// oaksLibrary/fbPushButton
//Funktionsblock för återfjädrande tryckknappar. För tex. förlängd drift aggregat. Om knapp återaktiveras innan tid löpt ut avvaktiveras utgång.
FUNCTION_BLOCK fbPushButton
VAR_INPUT
	bForceIndication : BOOL :=FALSE; //Tvångsstyrning indikering i tryckknapp
	bActiveTrig : BOOL := FALSE; // Läge på aktivering (V-tagg) ändras vid puls in på denna ingång. Är (V-tagg) till går den från och vise versa.
END_VAR

VAR_OUTPUT
	{attribute 'OPC.UA.DA' := '1'}
	V AT %M* : BOOL; //Aktiverad~wp:[trendoptions]i:14400, t:1
	{attribute 'OPC.UA.DA' := '1'}
	CMD AT %Q*: BOOL; //Indikering~wp:[trendoptions]i:14400, t:1
	{attribute 'OPC.UA.DA' := '1'}
	PV1 AT %M* : INT; //Återstående tid~wp:[unit]min[format]0
END_VAR

VAR
	bInput AT %I*: BOOL :=FALSE; //Ingång
	bMode: INT :=0; // Lägesindikering knapp 0=Avaktiverad funktion 1=Aktiverad knapp 2=Återaktiverad knapp (reset)
	bPulse: BOOL :=FALSE; // Startpuls
	tTime: TIME;
	rElapsed: REAL;
	rSetTime: REAL;
	fbResetTon : TON;
	fbTriggerPulse: TP;
	fbActivated: TP;
	fbCounter: CTU;
	fbResetFallingEdge: F_TRIG;	
END_VAR

VAR_INPUT PERSISTENT
	{attribute 'OPC.UA.DA' := '1'}
	SP1 AT %M*: INT :=120; //Frånslagsfördröjning~wp:[unit]min[format]0
	{attribute 'OPC.UA.DA' := '1'}
	M AT %M*: BOOL; //Handkörning~wp:[trendoptions]i:14400, t:1
END_VAR

	IF M THEN
		fbResetTon.IN := TRUE;
		IF fbResetTon.Q THEN
			M := FALSE;
		END_IF
	ELSE
		fbResetTon.IN := FALSE;
	END_IF
	fbResetTon.PT := T#0.5S;
	fbResetTon();

//Startpuls
fbTriggerPulse(IN:= bInput OR M OR bActiveTrig , PT:= T#0.5S , Q=> bPulse, ET=> );

//Återstånde tid
rElapsed := TIME_TO_REAL(fbActivated.ET);
rSetTime := TIME_TO_REAL(fbActivated.PT);
PV1 := REAL_TO_INT((rSetTime - rElapsed)/60000);

//Tidskonvertering till min->ms
tTime := INT_TO_TIME(SP1)*60000;

//Läge på knapp 
fbCounter(
	CU:= bPulse, 
	RESET:= fbCounter.Q OR fbResetFallingEdge.Q, 
	PV:= 2, 
	Q=> , 
	CV=>);

bMode := WORD_TO_INT(fbCounter.CV);

CASE bMode OF
0:
fbActivated.PT := T#0S;
1:
fbActivated.PT := tTime ;	
END_CASE
//Utgång
fbActivated(IN:= bMode=1, PT:=, Q=> V, ET=> );
CMD := V OR bForceIndication;
//Reset av funktion då tid löpt ut
fbResetFallingEdge(CLK:= fbActivated.Q , Q=> );

END_FUNCTION_BLOCK

// oaksLibrary/Regulatorer/Utökade regulatorer/fbAdvSequenceController2Stages
// Pi-regulator 2-sekvens
// För utökad kontroll av reglering:
// bPause fryser regulatorns läge
// bSync synkar regulatorns aktuella sekvens till sitt inställda rSync-värde
// udiInitSwDl är fördröjning innan byte av sekvens vid uppstart (om 0 funkar ej vald startsekvens om PV < SP)
// rSyncSeq[n] är synkvärde för resp sekvens
// rOffValSeq[n] är fast utsignal då bEnable = FALSE
{attribute 'initialize_on_call'}
FUNCTION_BLOCK fbAdvSequenceController2Stages
VAR_INPUT
	bEnable : BOOL; // Aktiverar reglering
	bPause : BOOL := FALSE; // Pausa regulator
	bSync : BOOL := FALSE; // Synkronisera aktuell sekvens till rSync
	udiInitSwDl : UDINT := 5; // Fördröjning för växling av sekvens vid uppstart (minst 1 om startsekvens ska gälla)	
	rProcessValue : REAL; // Aktuellt Ärvärde 
	rSetpoint : REAL; // Aktuellt börvärde. Önskas separat kylbörvärde för kylsekvenser se inputen rCoolSetpoint.
	{attribute 'initialize_on_call'}
	rCoolSetpoint : REFERENCE TO REAL := 0; //Om man önskar ha ett högre börvärde för kylsekvenser lägg denna här så väljs detta på de sekvenser där bActnSequenceX = TRUE. Lämnar man inputen tom körs rSetpoint på både kyl och värmesekvenser.
	iStartSequence : UDINT := 2; //Sekvens där regulator startar
	
	rMinSeq1 : REAL := 0; 
	rMaxSeq1 : REAL := 100; 
	rSyncSeq1 : REAL := 0;	//Synkvärde
	rOffValSeq1 : REAL := 0; //Utgång om ej bEnable
	bActnSequence1 : BOOL; // Gångriktning reglersekvens  (kylsekvens = TRUE)
	bBlockSequence1 : BOOL; // blockera denna sekvens kan användas exempelvis vid nattkyla
	rKpSequence1 : REAL; // Kp
	rKiSequence1 : UDINT; // Ki
	rDiSequence1 : UDINT; // D-tid (Derivata)
	rFDiSequence1 : UDINT; // Filter tid D (Derivata)
	rDzSequence1 : REAL :=0.1; //Dödzon
	
	rMinSeq2 : REAL := 0; 
	rMaxSeq2 : REAL := 100; 
	rSyncSeq2 : REAL := 0;	//Synkvärde
	rOffValSeq2 : REAL := 0; //Utgång om ej bEnable
	bActnSequence2 : BOOL; // Gångriktning reglersekvens  (kylsekvens = TRUE)
	bBlockSequence2 : BOOL; // blockera denna sekvens kan användas exempelvis vid nattkyla
	rKpSequence2 : REAL; // Kp
	rKiSequence2 : UDINT; // Ki
	rDiSequence2 : UDINT; // D-tid (Derivata)
	rFDiSequence2 : UDINT; // Filter tid D (Derivata)
	rDzSequence2 : REAL :=0.1; //Dödzon

	{attribute 'initialize_on_call'}
	rDevLimit : REFERENCE TO REAL := 0;
	{attribute 'pingroup' := 'DeviationAlarm'}
	bBlockHighAlarm : BOOL; // Blockera högtemplarm
	{attribute 'pingroup' := 'DeviationAlarm'}
	bBlockLowAlarm : BOOL; // Blockera lågtemplarm
	{attribute 'pingroup' := 'DeviationAlarm'}
	tAlarmDelay : TIME := T#5S; // larmfördröjning
END_VAR
VAR_OUTPUT
	rOutputSequence1 : REAL;  // regulatorsignal
	rOutputSequence2 : REAL;  // regulatorsignal
	{attribute 'pingroup' := 'DeviationAlarm'}
	bAlarmOutput : BOOL; //larmutgång
END_VAR
VAR
	rDevLimitInternal : REAL;
	fbDevAlarmPV: fbDevAlarm;
	rSetPointSequence1,rSetPointSequence2 : REAL; 	

	rTempMin,rTempMax : REAL; // tempvariabel för blockering av sekvenser 
	fbSeqLink01: Tc3_BA_Common.FB_BA_SeqLink;
	stSeqLink01 : Tc3_BA_Common.ST_BA_SeqLink;
	fbPidSeq: ARRAY[1..2] OF Tc3_BA_Common.FB_BA_SeqCtrl;
	iStartSequenceInternal : UDINT := 2;
	
	fbEdgeEnable : fbEdge;
END_VAR

fbEdgeEnable(anyInput := bEnable);
IF fbEdgeEnable.bEdgeF THEN bSync := TRUE; END_IF	

fbDevAlarmPV(
	tAlarmDelay:=tAlarmDelay , 
	bAutoReset:=TRUE , 
	bAlarmOutput=>bAlarmOutput , 
	bEnable:=bEnable AND mDevAlarmCheck(), 
	rProcessValue:=rProcessValue , 
	rSetPoint:=rSetpoint , 
	rDevLimit:=rDevLimitInternal , 
	bBlockHighAlarm:=bBlockHighAlarm , 
	bBlockLowAlarm:=bBlockLowAlarm );

	IF iStartSequence > 0 AND iStartSequence < 3 THEN
	 iStartSequenceInternal	 := 3 - iStartSequence;
	END_IF;

IF NOT bPause THEN
	fbSeqLink01(
	bEn:= bEnable, 
	udiSttCtrl:=iStartSequenceInternal , 
	udiIniSwiOvrDly_sec:= udiInitSwDl, 
	rX:= rProcessValue, 
	stSeqLink:=stSeqLink01 , 
	udiCurCtrl=> , 
	bSeqActv=> , 
	bNotRead=> , 
	bNoneOp=> , 
	udiRemTiIniSwiOvrDly_sec=> , 
	bErr=> , 
	sErrDescr=> );
	
	IF bBlockSequence1 THEN
		rTempMin := 0;
		rTempMax := 0;
	ELSE
		rTempMin := rMinSeq1;
		rTempMax := rMaxSeq1;
	END_IF
	rSetPointSequence1 := mCoolSetpointCheck(bActnSequence1);
	fbPidSeq[1](
	bEn:=bEnable , 
	rW:= rSetPointSequence1, 
	rX:=rProcessValue , 
	udiOpMode:= , 
	bActn:=bActnSequence1 , 
	rKp:= rKpSequence1, 
	udiTn_ms:=rKiSequence1*1000 , 
	udiTv_ms:=rDiSequence1*1000 , 
	udiTd_ms:=rFDiSequence1*1000 , 
	rYMax:=rTempMax , 
	rYMin:=rTempMin , 
	rNZ:= rDzSequence1, 
	udiCycCl:= , 
	bSync:= bSync, 
	rSync:= rSyncSeq1, 
	rYSeqInit:= rSyncSeq1, 
	udiMyNum:= 2, 
	stSeqLink:=stSeqLink01 , 
	rY=> rOutputSequence1, 
	rE=> , 
	bErr=> , 
	sErrDescr=> );
	
	IF bBlockSequence2 THEN
		rTempMin := 0;
		rTempMax := 0;
	ELSE
		rTempMin := rMinSeq2;
		rTempMax := rMaxSeq2;
	END_IF
	rSetPointSequence2 := mCoolSetpointCheck(bActnSequence2);
	fbPidSeq[2](
	bEn:=bEnable , 
	rW:= rSetPointSequence2, 
	rX:= rProcessValue, 
	udiOpMode:= , 
	bActn:= bActnSequence2, 
	rKp:= rKpSequence2, 
	udiTn_ms:=rKiSequence2*1000 , 
	udiTv_ms:=rDiSequence2*1000  , 
	udiTd_ms:=rFDiSequence2*1000 , 
	rYMax:=rTempMax , 
	rYMin:=rTempMin , 
	rNZ:= rDzSequence2, 
	udiCycCl:= , 
	bSync:= bSync, 
	rSync:= rSyncSeq2, 
	rYSeqInit:= rSyncSeq2, 
	udiMyNum:= 1, 
	stSeqLink:= stSeqLink01, 
	rY=> rOutputSequence2, 
	rE=> , 
	bErr=> , 
	sErrDescr=> );
	
	bSync := FALSE;	
END_IF;

IF NOT bEnable THEN
	rOutputSequence1 := rOffValSeq1;
	rOutputSequence2 := rOffValSeq2;
END_IF

// Publik metod för att kolla ifall det finns någon kylsekvens i regleringen. Kan exempelvis användas för att blockera högavvikelselarm vid hög utetemperatur då kylsekvens saknas.
METHOD PUBLIC mContainsCoolingSequence : BOOL
mContainsCoolingSequence := bActnSequence1 OR bActnSequence2;
END_METHOD

// Metod för att kolla ifall det är en kylsekvens och om det i sådant fall är något knutet på rCoolSetpoint
METHOD PRIVATE mCoolSetpointCheck : REAL // Valt börvärde
VAR_INPUT
	bActn : BOOL; // Koll av gångriktning
END_VAR
IF NOT bActn THEN
	mCoolSetpointCheck := rSetpoint;
ELSE
	IF __ISVALIDREF(rCoolSetpoint) THEN 
		mCoolSetpointCheck := rCoolSetpoint;
	ELSE
		mCoolSetpointCheck := rSetpoint;
	END_IF
END_IF
END_METHOD

// Kolla ifall något är knutet på inputen rDevLimit. Är inget knutet där inaktiveras avvikelselarmet.
METHOD PRIVATE mDevAlarmCheck : BOOL // Valt börvärde
IF __ISVALIDREF(rDevLimit) THEN 
	mDevAlarmCheck := TRUE;
	rDevLimitInternal := rDevLimit;
ELSE
	mDevAlarmCheck := FALSE;
END_IF
END_METHOD

END_FUNCTION_BLOCK

// oaksLibrary/Regulatorer/Utökade regulatorer/fbAdvSequenceController3Stages
// Pi-regulator 3-sekvens
// För utökad kontroll av reglering:
// bPause fryser regulatorns läge
// bSync synkar regulatorns aktuella sekvens till sitt inställda rSync-värde
// udiInitSwDl är fördröjning innan byte av sekvens vid uppstart (om 0 funkar ej vald startsekvens om PV < SP)
// rSyncSeq[n] är synkvärde för resp sekvens
// rOffValSeq[n] är fast utsignal då bEnable = FALSE
{attribute 'initialize_on_call'}
FUNCTION_BLOCK fbAdvSequenceController3Stages
VAR_INPUT
	bEnable : BOOL; // Aktiverar reglering (toggla för att reset:a regulator)
	bPause : BOOL := FALSE; // Pausa regulator
	bSync : BOOL := FALSE; // Synkronisera aktuell sekvens till rSync
	udiInitSwDl : UDINT := 5; // Fördröjning för växling av sekvens vid uppstart (minst 1 om startsekvens ska gälla)	
	rProcessValue : REAL; // Aktuellt Ärvärde 
	rSetpoint : REAL; // Aktuellt börvärde. Önskas separat kylbörvärde för kylsekvenser se inputen rCoolSetpoint.
	{attribute 'initialize_on_call'}
	rCoolSetpoint : REFERENCE TO REAL; //Om man önskar ha ett högre börvärde för kylsekvenser lägg denna här så väljs detta på de sekvenser där bActnSequenceX = TRUE. Lämnar man inputen tom körs rSetpoint på både kyl och värmesekvenser.
	iStartSequence : UDINT :=3; //Sekvens där regulator startar
	
	rMinSeq1 : REAL := 0;	//Min utsignal
	rMaxSeq1 : REAL := 100;	//Max utsignal
	rSyncSeq1 : REAL := 0;	//Synkvärde
	rOffValSeq1 : REAL := 0; //Utgång om ej bEnable
	bActnSequence1 : BOOL; // Gångriktning reglersekvens  (kylsekvens = TRUE)
	bBlockSequence1 : BOOL; // blockera denna sekvens kan användas exempelvis vid nattkyla
	rKpSequence1 : REAL; // Kp
	rKiSequence1 : UDINT; // Ki
	rDiSequence1 : UDINT; // D-tid (Derivata)
	rFDiSequence1 : UDINT; // Filter tid D (Derivata)
	rDzSequence1 : REAL :=0.1; //Dödzon
	
	rMinSeq2 : REAL := 0; 
	rMaxSeq2 : REAL := 100;
	rSyncSeq2 : REAL := 0;
	rOffValSeq2 : REAL := 0; //Utgång om ej bEnable
	bActnSequence2 : BOOL; // Gångriktning reglersekvens  (kylsekvens = TRUE)
	bBlockSequence2 : BOOL; // blockera denna sekvens kan användas exempelvis vid nattkyla
	rKpSequence2 : REAL; // Kp
	rKiSequence2 : UDINT; // Ki
	rDiSequence2 : UDINT; // D-tid (Derivata)
	rFDiSequence2 : UDINT; // Filter tid D (Derivata)
	rDzSequence2 : REAL :=0.1; //Dödzon
	
	rMinSeq3 : REAL := 0; 
	rMaxSeq3 : REAL := 100;
	rSyncSeq3 : REAL := 0;
	rOffValSeq3 : REAL := 0; //Utgång om ej bEnable
	bActnSequence3 : BOOL; // Gångriktning reglersekvens  (kylsekvens = TRUE)
	bBlockSequence3 : BOOL; // blockera denna sekvens kan användas exempelvis vid nattkyla
	rKpSequence3 : REAL; // Kp
	rKiSequence3 : UDINT; // Ki
	rDiSequence3 : UDINT; // D-tid (Derivata)
	rFDiSequence3 : UDINT; // Filter tid D (Derivata)
	rDzSequence3 : REAL :=0.1; //Dödzon
	
	{attribute 'pingroup' := 'DeviationAlarm'}
	{attribute 'initialize_on_call'}
	rDevLimit : REFERENCE TO REAL := 0;
	{attribute 'pingroup' := 'DeviationAlarm'}
	bBlockHighAlarm : BOOL; // Blockera högtemplarm
	{attribute 'pingroup' := 'DeviationAlarm'}
	bBlockLowAlarm : BOOL; // Blockera lågtemplarm
	{attribute 'pingroup' := 'DeviationAlarm'}
	tAlarmDelay : TIME := T#5S; // larmfördröjning
END_VAR
VAR_OUTPUT
	rOutputSequence1 : REAL;  // regulatorsignal
	rOutputSequence2 : REAL;  // regulatorsignal
	rOutputSequence3 : REAL;  // regulatorsignal
	{attribute 'pingroup' := 'DeviationAlarm'}
	bAlarmOutput : BOOL; //larmutgång
END_VAR
VAR
	rDevLimitInternal : REAL;
	fbDevAlarmPV: fbDevAlarm;
	rSetPointSequence1,rSetPointSequence2,rSetPointSequence3 : REAL; 		

	rTempMin,rTempMax : REAL; // tempvariabel för blockering av sekvenser 
	fbSeqLink01: Tc3_BA_Common.FB_BA_SeqLink;
	stSeqLink01 : Tc3_BA_Common.ST_BA_SeqLink;
	fbPidSeq: ARRAY[1..3] OF Tc3_BA_Common.FB_BA_SeqCtrl;
	iStartSequenceInternal : UDINT := 3;
	
	fbEdgeEnable : fbEdge;
END_VAR

fbEdgeEnable(anyInput := bEnable);
IF fbEdgeEnable.bEdgeF THEN bSync := TRUE; END_IF

fbDevAlarmPV(
tAlarmDelay:=tAlarmDelay , 
bAutoReset:=TRUE , 
bAlarmOutput=>bAlarmOutput , 
bEnable:=bEnable AND mDevAlarmCheck(), 
rProcessValue:=rProcessValue , 
rSetPoint:=rSetpoint , 
rDevLimit:=rDevLimitInternal , 
bBlockHighAlarm:=bBlockHighAlarm , 
bBlockLowAlarm:=bBlockLowAlarm );

IF iStartSequence > 0 AND iStartSequence < 4 THEN
 iStartSequenceInternal	 := 4 - iStartSequence;
END_IF;
		
IF NOT bPause THEN	
	fbSeqLink01(
	bEn:= bEnable, 
	udiSttCtrl:= iStartSequenceInternal, 
	udiIniSwiOvrDly_sec:= udiInitSwDl, 
	rX:= rProcessValue, 
	stSeqLink:=stSeqLink01 , 
	udiCurCtrl=> , 
	bSeqActv=> , 
	bNotRead=> , 
	bNoneOp=> , 
	udiRemTiIniSwiOvrDly_sec=> , 
	bErr=> , 
	sErrDescr=> );
	
	IF bBlockSequence1 THEN
		rTempMin := 0;
		rTempMax := 0;
	ELSE
		rTempMin := rMinSeq1;
		rTempMax := rMaxSeq1;
	END_IF
	rSetPointSequence1 := mCoolSetpointCheck(bActnSequence1);
	fbPidSeq[1](
	bEn:=bEnable , 
	rW:= rSetPointSequence1, 
	rX:=rProcessValue , 
	udiOpMode:= , 
	bActn:=bActnSequence1 , 
	rKp:= rKpSequence1, 
	udiTn_ms:=rKiSequence1*1000 , 
	udiTv_ms:=rDiSequence1*1000 , 
	udiTd_ms:=rFDiSequence1*1000 , 
	rYMax:=rTempMax , 
	rYMin:= rTempMin, 
	rNZ:= rDzSequence1, 
	udiCycCl:= , 
	bSync:= bSync, 
	rSync:= rSyncSeq1, 
	rYSeqInit:= rSyncSeq1, 
	udiMyNum:= 3, 
	stSeqLink:=stSeqLink01 , 
	rY=> rOutputSequence1, 
	rE=> , 
	bErr=> , 
	sErrDescr=> );
	
	IF bBlockSequence2 THEN
		rTempMin := 0;
		rTempMax := 0;
	ELSE
		rTempMin := rMinSeq2;
		rTempMax := rMaxSeq2;
	END_IF
	rSetPointSequence2 := mCoolSetpointCheck(bActnSequence2);
	fbPidSeq[2](
	bEn:=bEnable , 
	rW:= rSetPointSequence2, 
	rX:= rProcessValue, 
	udiOpMode:= , 
	bActn:= bActnSequence2, 
	rKp:= rKpSequence2, 
	udiTn_ms:=rKiSequence2*1000 , 
	udiTv_ms:=rDiSequence2*1000 , 
	udiTd_ms:=rFDiSequence2*1000 , 
	rYMax:= rTempMax, 
	rYMin:=rTempMin , 
	rNZ:= rDzSequence2, 
	udiCycCl:= , 
	bSync:= bSync,  
	rSync:= rSyncSeq2, 
	rYSeqInit:= rSyncSeq2, 
	udiMyNum:= 2, 
	stSeqLink:= stSeqLink01, 
	rY=> rOutputSequence2, 
	rE=> , 
	bErr=> , 
	sErrDescr=> );
	
	IF bBlockSequence3 THEN
		rTempMin := 0;
		rTempMax := 0;
	ELSE
		rTempMin := rMinSeq3;
		rTempMax := rMaxSeq3;
	END_IF
	rSetPointSequence3 := mCoolSetpointCheck(bActnSequence3);
	fbPidSeq[3](
	bEn:=bEnable , 
	rW:= rSetPointSequence3, 
	rX:= rProcessValue, 
	udiOpMode:= , 
	bActn:= bActnSequence3, 
	rKp:= rKpSequence3, 
	udiTn_ms:=rKiSequence3*1000 , 
	udiTv_ms:=rDiSequence3*1000 , 
	udiTd_ms:=rFDiSequence3*1000 , 
	rYMax:=rTempMax , 
	rYMin:= rTempMin, 
	rNZ:= rDzSequence3, 
	udiCycCl:= , 
	bSync:= bSync, 
	rSync:= rSyncSeq3, 
	rYSeqInit:= rSyncSeq3, 
	udiMyNum:= 1, 
	stSeqLink:= stSeqLink01, 
	rY=> rOutputSequence3, 
	rE=> , 
	bErr=> , 
	sErrDescr=> );
	
	bSync := FALSE;	
END_IF;

IF NOT bEnable THEN
	rOutputSequence1 := rOffValSeq1;
	rOutputSequence2 := rOffValSeq2;
	rOutputSequence3 := rOffValSeq3;
END_IF

// Publik metod för att kolla ifall det finns någon kylsekvens i regleringen. Kan exempelvis användas för att blockera högavvikelselarm vid hög utetemperatur då kylsekvens saknas.
METHOD PUBLIC mContainsCoolingSequence : BOOL
mContainsCoolingSequence := bActnSequence1 OR bActnSequence2 OR bActnSequence3;
END_METHOD

// Metod för att kolla ifall det är en kylsekvens och om det i sådant fall är något knutet på rCoolSetpoint
METHOD PRIVATE mCoolSetpointCheck : REAL // Valt börvärde
VAR_INPUT
	bActn : BOOL; // Koll av gångriktning
END_VAR
IF NOT bActn THEN
	mCoolSetpointCheck := rSetpoint;
ELSE
	IF __ISVALIDREF(rCoolSetpoint) THEN 
		mCoolSetpointCheck := rCoolSetpoint;
	ELSE
		mCoolSetpointCheck := rSetpoint;
	END_IF
END_IF
END_METHOD

// Kolla ifall något är knutet på inputen rDevLimit. Är inget knutet där inaktiveras avvikelselarmet.
METHOD PRIVATE mDevAlarmCheck : BOOL // Valt börvärde
IF __ISVALIDREF(rDevLimit) THEN 
	mDevAlarmCheck := TRUE;
	rDevLimitInternal := rDevLimit;
ELSE
	mDevAlarmCheck := FALSE;
END_IF
END_METHOD

END_FUNCTION_BLOCK

// oaksLibrary/Regulatorer/Utökade regulatorer/fbAdvSequenceController4Stages
// Pi-regulator 4-sekvens
// För utökad kontroll av reglering:
// bPause fryser regulatorns läge
// bSync synkar regulatorns aktuella sekvens till sitt inställda rSync-värde
// udiInitSwDl är fördröjning innan byte av sekvens vid uppstart (om 0 funkar ej vald startsekvens om PV < SP)
// rSyncSeq[n] är synkvärde för resp sekvens
// rOffValSeq[n] är fast utsignal då bEnable = FALSE
{attribute 'initialize_on_call'}
FUNCTION_BLOCK fbAdvSequenceController4Stages
VAR_INPUT
	bEnable : BOOL; // Aktiverar reglering (toggla för att reset:a regulator)
	bPause : BOOL := FALSE; // Pausa regulator
	bSync : BOOL := FALSE; // Synkronisera aktuell sekvens till rSync
	udiInitSwDl : UDINT := 5; // Fördröjning för växling av sekvens vid uppstart (minst 1 om startsekvens ska gälla)	
	rProcessValue : REAL; // Aktuellt Ärvärde 
	rSetpoint : REAL; // Aktuellt börvärde. Önskas separat kylbörvärde för kylsekvenser se inputen rCoolSetpoint.
	{attribute 'initialize_on_call'}
	rCoolSetpoint : REFERENCE TO REAL; //Om man önskar ha ett högre börvärde för kylsekvenser lägg denna här så väljs detta på de sekvenser där bActnSequenceX = TRUE. Lämnar man inputen tom körs rSetpoint på både kyl och värmesekvenser.
	iStartSequence : UDINT :=3; //Sekvens där regulator startar
	
	rMinSeq1 : REAL := 0;	//Min utsignal
	rMaxSeq1 : REAL := 100;	//Max utsignal
	rSyncSeq1 : REAL := 0;	//Synkvärde
	rOffValSeq1 : REAL := 0; //Utgång om ej bEnable
	bActnSequence1 : BOOL; // Gångriktning reglersekvens  (kylsekvens = TRUE)
	bBlockSequence1 : BOOL; // blockera denna sekvens kan användas exempelvis vid nattkyla
	rKpSequence1 : REAL; // Kp
	rKiSequence1 : UDINT; // Ki
	rDiSequence1 : UDINT; // D-tid (Derivata)
	rFDiSequence1 : UDINT; // Filter tid D (Derivata)
	rDzSequence1 : REAL :=0.1; //Dödzon
	
	rMinSeq2 : REAL := 0; 
	rMaxSeq2 : REAL := 100;
	rSyncSeq2 : REAL := 0;
	rOffValSeq2 : REAL := 0; //Utgång om ej bEnable
	bActnSequence2 : BOOL; // Gångriktning reglersekvens  (kylsekvens = TRUE)
	bBlockSequence2 : BOOL; // blockera denna sekvens kan användas exempelvis vid nattkyla
	rKpSequence2 : REAL; // Kp
	rKiSequence2 : UDINT; // Ki
	rDiSequence2 : UDINT; // D-tid (Derivata)
	rFDiSequence2 : UDINT; // Filter tid D (Derivata)
	rDzSequence2 : REAL :=0.1; //Dödzon
	
	rMinSeq3 : REAL := 0; 
	rMaxSeq3 : REAL := 100;
	rSyncSeq3 : REAL := 0;
	rOffValSeq3 : REAL := 0; //Utgång om ej bEnable
	bActnSequence3 : BOOL; // Gångriktning reglersekvens  (kylsekvens = TRUE)
	bBlockSequence3 : BOOL; // blockera denna sekvens kan användas exempelvis vid nattkyla
	rKpSequence3 : REAL; // Kp
	rKiSequence3 : UDINT; // Ki
	rDiSequence3 : UDINT; // D-tid (Derivata)
	rFDiSequence3 : UDINT; // Filter tid D (Derivata)
	rDzSequence3 : REAL :=0.1; //Dödzon
	
	rMinSeq4 : REAL := 0; 
	rMaxSeq4 : REAL := 100;
	rSyncSeq4 : REAL := 0;
	rOffValSeq4 : REAL := 0; //Utgång om ej bEnable
	bActnSequence4 : BOOL; // Gångriktning reglersekvens  (kylsekvens = TRUE)
	bBlockSequence4 : BOOL; // blockera denna sekvens kan användas exempelvis vid nattkyla
	rKpSequence4 : REAL; // Kp
	rKiSequence4 : UDINT; // Ki
	rDiSequence4 : UDINT; // D-tid (Derivata)
	rFDiSequence4 : UDINT; // Filter tid D (Derivata)
	rDzSequence4 : REAL :=0.1; //Dödzon
	
	{attribute 'pingroup' := 'DeviationAlarm'}
	{attribute 'initialize_on_call'}
	rDevLimit : REFERENCE TO REAL := 0;
	{attribute 'pingroup' := 'DeviationAlarm'}
	bBlockHighAlarm : BOOL; // Blockera högtemplarm
	{attribute 'pingroup' := 'DeviationAlarm'}
	bBlockLowAlarm : BOOL; // Blockera lågtemplarm
	{attribute 'pingroup' := 'DeviationAlarm'}
	tAlarmDelay : TIME := T#5S; // larmfördröjning
END_VAR
VAR_OUTPUT
	rY : REAL; // Utsignal huvudregulator
	rOutputSequence1 : REAL;  // regulatorsignal
	rOutputSequence2 : REAL;  // regulatorsignal
	rOutputSequence3 : REAL;  // regulatorsignal
	rOutputSequence4 : REAL;  // regulatorsignal
	{attribute 'pingroup' := 'DeviationAlarm'}
	bAlarmOutput : BOOL; //larmutgång
END_VAR
VAR
	rDevLimitInternal : REAL;
	fbDevAlarmPV: fbDevAlarm;
	rSetPointSequence1,rSetPointSequence2,rSetPointSequence3,rSetPointSequence4 : REAL; 	
	rTempMin,rTempMax : REAL; // tempvariabel för blockering av sekvenser 
	fbSeqLink01: Tc3_BA_Common.FB_BA_SeqLink;
	stSeqLink01 : Tc3_BA_Common.ST_BA_SeqLink;
	fbPidSeq: ARRAY[1..4] OF Tc3_BA_Common.FB_BA_SeqCtrl;
	iStartSequenceInternal : UDINT := 3;
	
	fbEdgeEnable : fbEdge;
END_VAR

fbEdgeEnable(anyInput := bEnable);
IF fbEdgeEnable.bEdgeF THEN bSync := TRUE; END_IF

	fbDevAlarmPV(
	tAlarmDelay:=tAlarmDelay , 
	bAutoReset:=TRUE , 
	bAlarmOutput=>bAlarmOutput , 
	bEnable:=bEnable AND mDevAlarmCheck(), 
	rProcessValue:=rProcessValue , 
	rSetPoint:=rSetpoint , 
	rDevLimit:=rDevLimitInternal , 
	bBlockHighAlarm:=bBlockHighAlarm , 
	bBlockLowAlarm:=bBlockLowAlarm );

	IF iStartSequence > 0 AND iStartSequence < 5 THEN
	 iStartSequenceInternal	 := 5 - iStartSequence;
	END_IF;
		
IF NOT bPause THEN		
	fbSeqLink01(
	bEn:= bEnable, 
	udiSttCtrl:= iStartSequenceInternal, 
	udiIniSwiOvrDly_sec:= udiInitSwDl, 
	rX:= rProcessValue, 
	stSeqLink:=stSeqLink01 , 
	udiCurCtrl=> , 
	bSeqActv=> , 
	bNotRead=> , 
	bNoneOp=> , 
	udiRemTiIniSwiOvrDly_sec=> , 
	bErr=> , 
	sErrDescr=> );
		
	IF bBlockSequence1 THEN
		rTempMin := 0;
		rTempMax := 0;
	ELSE
		rTempMin := rMinSeq1;
		rTempMax := rMaxSeq1;
	END_IF
	rSetPointSequence1 := mCoolSetpointCheck(bActnSequence1);
	fbPidSeq[1](
	bEn:=bEnable , 
	rW:= rSetPointSequence1, 
	rX:=rProcessValue , 
	udiOpMode:= , 
	bActn:=bActnSequence1 , 
	rKp:= rKpSequence1, 
	udiTn_ms:=rKiSequence1*1000 , 
	udiTv_ms:=rDiSequence1*1000 , 
	udiTd_ms:=rFDiSequence1*1000 , 
	rYMax:=rTempMax , 
	rYMin:=rTempMin, 
	rNZ:= rDzSequence1, 
	udiCycCl:= , 
	bSync:= bSync, 
	rSync:= rSyncSeq1, 
	rYSeqInit:= rSyncSeq1, 
	udiMyNum:= 4, 
	stSeqLink:=stSeqLink01 , 
	rY=> rOutputSequence1, 
	rE=> , 
	bErr=> , 
	sErrDescr=> );
	
	IF bBlockSequence2 THEN
		rTempMin := 0;
		rTempMax := 0;
	ELSE
		rTempMin := rMinSeq2;
		rTempMax := rMaxSeq2;
	END_IF
	rSetPointSequence2 := mCoolSetpointCheck(bActnSequence2);
	fbPidSeq[2](
	bEn:=bEnable , 
	rW:= rSetPointSequence2, 
	rX:= rProcessValue, 
	udiOpMode:= , 
	bActn:= bActnSequence2, 
	rKp:= rKpSequence2, 
	udiTn_ms:=rKiSequence2*1000 , 
	udiTv_ms:=rDiSequence2*1000 , 
	udiTd_ms:=rFDiSequence2*1000 , 
	rYMax:= rTempMax, 
	rYMin:=rTempMin , 
	rNZ:= rDzSequence2, 
	udiCycCl:= , 
	bSync:= bSync, 
	rSync:= rSyncSeq2, 
	rYSeqInit:= rSyncSeq2, 
	udiMyNum:= 3, 
	stSeqLink:= stSeqLink01, 
	rY=> rOutputSequence2, 
	rE=> , 
	bErr=> , 
	sErrDescr=> );
	
	IF bBlockSequence3 THEN
		rTempMin := 0;
		rTempMax := 0;
	ELSE
		rTempMin := rMinSeq3;
		rTempMax := rMaxSeq3;
	END_IF
	rSetPointSequence3 := mCoolSetpointCheck(bActnSequence3);
	fbPidSeq[3](
	bEn:=bEnable , 
	rW:= rSetPointSequence3, 
	rX:= rProcessValue, 
	udiOpMode:= , 
	bActn:= bActnSequence3, 
	rKp:= rKpSequence3, 
	udiTn_ms:=rKiSequence3*1000 , 
	udiTv_ms:=rDiSequence3*1000 , 
	udiTd_ms:=rFDiSequence3*1000 , 
	rYMax:=rTempMax , 
	rYMin:= rTempMin, 
	rNZ:= rDzSequence3, 
	udiCycCl:= , 
	bSync:= bSync, 
	rSync:= rSyncSeq3, 
	rYSeqInit:= rSyncSeq3, 
	udiMyNum:= 2, 
	stSeqLink:= stSeqLink01, 
	rY=> rOutputSequence3, 
	rE=> , 
	bErr=> , 
	sErrDescr=> );
	
	IF bBlockSequence4 THEN
		rTempMin := 0;
		rTempMax := 0;
	ELSE
		rTempMin := rMinSeq4;
		rTempMax := rMaxSeq4;
	END_IF
	rSetPointSequence4 := mCoolSetpointCheck(bActnSequence4);
	fbPidSeq[4](
	bEn:=bEnable , 
	rW:= rSetPointSequence4, 
	rX:= rProcessValue, 
	udiOpMode:= , 
	bActn:= bActnSequence4, 
	rKp:= rKpSequence4, 
	udiTn_ms:=rKiSequence4*1000 , 
	udiTv_ms:=rDiSequence4*1000 , 
	udiTd_ms:=rFDiSequence4*1000 , 
	rYMax:=rTempMax , 
	rYMin:= rTempMin, 
	rNZ:= rDzSequence4, 
	udiCycCl:= , 
	bSync:= bSync, 
	rSync:= rSyncSeq4, 
	rYSeqInit:= rSyncSeq4, 
	udiMyNum:= 1, 
	stSeqLink:= stSeqLink01, 
	rY=> rOutputSequence4, 
	rE=> , 
	bErr=> , 
	sErrDescr=> );
	
	bSync := FALSE;	
END_IF

IF NOT bEnable THEN
	rOutputSequence1 := rOffValSeq1;
	rOutputSequence2 := rOffValSeq2;
	rOutputSequence3 := rOffValSeq3;
	rOutputSequence4 := rOffValSeq4;
END_IF

// Publik metod för att kolla ifall det finns någon kylsekvens i regleringen. Kan exempelvis användas för att blockera högavvikelselarm vid hög utetemperatur då kylsekvens saknas.
METHOD PUBLIC mContainsCoolingSequence : BOOL
mContainsCoolingSequence := bActnSequence1 OR bActnSequence2 OR bActnSequence3 OR bActnSequence4;
END_METHOD

// Metod för att kolla ifall det är en kylsekvens och om det i sådant fall är något knutet på rCoolSetpoint
METHOD PRIVATE mCoolSetpointCheck : REAL // Valt börvärde
VAR_INPUT
	bActn : BOOL; // Koll av gångriktning
END_VAR
IF NOT bActn THEN
	mCoolSetpointCheck := rSetpoint;
ELSE
	IF __ISVALIDREF(rCoolSetpoint) THEN 
		mCoolSetpointCheck := rCoolSetpoint;
	ELSE
		mCoolSetpointCheck := rSetpoint;
	END_IF
END_IF
END_METHOD

// Kolla ifall något är knutet på inputen rDevLimit. Är inget knutet där inaktiveras avvikelselarmet.
METHOD PRIVATE mDevAlarmCheck : BOOL // Valt börvärde
IF __ISVALIDREF(rDevLimit) THEN 
	mDevAlarmCheck := TRUE;
	rDevLimitInternal := rDevLimit;
ELSE
	mDevAlarmCheck := FALSE;
END_IF
END_METHOD

END_FUNCTION_BLOCK

// oaksLibrary/Regulatorer/Utökade regulatorer/fbAdvSequenceController5Stages
// Pi-regulator 5-sekvens
// För utökad kontroll av reglering:
// bPause fryser regulatorns läge
// bSync synkar regulatorns aktuella sekvens till sitt inställda rSync-värde
// udiInitSwDl är fördröjning innan byte av sekvens vid uppstart (om 0 funkar ej vald startsekvens om PV < SP)
// rSyncSeq[n] är synkvärde för resp sekvens
// rOffValSeq[n] är fast utsignal då bEnable = FALSE
{attribute 'initialize_on_call'}
FUNCTION_BLOCK fbAdvSequenceController5Stages
VAR_INPUT
	bEnable : BOOL; // Aktiverar reglering (toggla för att reset:a regulator)
	bPause : BOOL := FALSE; // Pausa regulator
	bSync : BOOL := FALSE; // Synkronisera aktuell sekvens till rSync
	udiInitSwDl : UDINT := 5; // Fördröjning för växling av sekvens vid uppstart (minst 1 om startsekvens ska gälla)	
	rProcessValue : REAL; // Aktuellt Ärvärde 
	rSetpoint : REAL; // Aktuellt börvärde. Önskas separat kylbörvärde för kylsekvenser se inputen rCoolSetpoint.
	{attribute 'initialize_on_call'}
	rCoolSetpoint : REFERENCE TO REAL; //Om man önskar ha ett högre börvärde för kylsekvenser lägg denna här så väljs detta på de sekvenser där bActnSequenceX = TRUE. Lämnar man inputen tom körs rSetpoint på både kyl och värmesekvenser.
	iStartSequence : UDINT :=3; //Sekvens där regulator startar
	
	rMinSeq1 : REAL := 0;	//Min utsignal
	rMaxSeq1 : REAL := 100;	//Max utsignal
	rSyncSeq1 : REAL := 0;	//Synkvärde
	rOffValSeq1 : REAL := 0; //Utgång om ej bEnable
	bActnSequence1 : BOOL; // Gångriktning reglersekvens  (kylsekvens = TRUE)
	bBlockSequence1 : BOOL; // blockera denna sekvens kan användas exempelvis vid nattkyla
	rKpSequence1 : REAL; // Kp
	rKiSequence1 : UDINT; // Ki
	rDiSequence1 : UDINT; // D-tid (Derivata)
	rFDiSequence1 : UDINT; // Filter tid D (Derivata)
	rDzSequence1 : REAL :=0.1; //Dödzon
	
	rMinSeq2 : REAL := 0; 
	rMaxSeq2 : REAL := 100;
	rSyncSeq2 : REAL := 0;
	rOffValSeq2 : REAL := 0; //Utgång om ej bEnable
	bActnSequence2 : BOOL; // Gångriktning reglersekvens  (kylsekvens = TRUE)
	bBlockSequence2 : BOOL; // blockera denna sekvens kan användas exempelvis vid nattkyla
	rKpSequence2 : REAL; // Kp
	rKiSequence2 : UDINT; // Ki
	rDiSequence2 : UDINT; // D-tid (Derivata)
	rFDiSequence2 : UDINT; // Filter tid D (Derivata)
	rDzSequence2 : REAL :=0.1; //Dödzon
	
	rMinSeq3 : REAL := 0; 
	rMaxSeq3 : REAL := 100;
	rSyncSeq3 : REAL := 0;
	rOffValSeq3 : REAL := 0; //Utgång om ej bEnable
	bActnSequence3 : BOOL; // Gångriktning reglersekvens  (kylsekvens = TRUE)
	bBlockSequence3 : BOOL; // blockera denna sekvens kan användas exempelvis vid nattkyla
	rKpSequence3 : REAL; // Kp
	rKiSequence3 : UDINT; // Ki
	rDiSequence3 : UDINT; // D-tid (Derivata)
	rFDiSequence3 : UDINT; // Filter tid D (Derivata)
	rDzSequence3 : REAL :=0.1; //Dödzon
	
	rMinSeq4 : REAL := 0; 
	rMaxSeq4 : REAL := 100;
	rSyncSeq4 : REAL := 0;	//Synkvärde
	rOffValSeq4 : REAL := 0; //Utgång om ej bEnable
	bActnSequence4 : BOOL; // Gångriktning reglersekvens  (kylsekvens = TRUE)
	bBlockSequence4 : BOOL; // blockera denna sekvens kan användas exempelvis vid nattkyla
	rKpSequence4 : REAL; // Kp
	rKiSequence4 : UDINT; // Ki
	rDiSequence4 : UDINT; // D-tid (Derivata)
	rFDiSequence4 : UDINT; // Filter tid D (Derivata)
	rDzSequence4 : REAL :=0.1; //Dödzon
	
	rMinSeq5 : REAL := 0; 
	rMaxSeq5 : REAL := 100;
	rSyncSeq5 : REAL := 0;	//Synkvärde
	rOffValSeq5 : REAL := 0; //Utgång om ej bEnable
	bActnSequence5 : BOOL; // Gångriktning reglersekvens  (kylsekvens = TRUE)
	bBlockSequence5 : BOOL; // blockera denna sekvens kan användas exempelvis vid nattkyla
	rKpSequence5 : REAL; // Kp
	rKiSequence5 : UDINT; // Ki
	rDiSequence5 : UDINT; // D-tid (Derivata)
	rFDiSequence5 : UDINT; // Filter tid D (Derivata)
	rDzSequence5 : REAL :=0.1; //Dödzon
	
	{attribute 'pingroup' := 'DeviationAlarm'}
	{attribute 'initialize_on_call'}
	rDevLimit : REFERENCE TO REAL := 0;
	{attribute 'pingroup' := 'DeviationAlarm'}
	bBlockHighAlarm : BOOL; // Blockera högtemplarm
	{attribute 'pingroup' := 'DeviationAlarm'}
	bBlockLowAlarm : BOOL; // Blockera lågtemplarm
	{attribute 'pingroup' := 'DeviationAlarm'}
	tAlarmDelay : TIME := T#5S; // larmfördröjning
END_VAR
VAR_OUTPUT
	rY : REAL; // Utsignal huvudregulator
	rOutputSequence1 : REAL;  // regulatorsignal
	rOutputSequence2 : REAL;  // regulatorsignal
	rOutputSequence3 : REAL;  // regulatorsignal
	rOutputSequence4 : REAL;  // regulatorsignal
	rOutputSequence5 : REAL;  // regulatorsignal
	{attribute 'pingroup' := 'DeviationAlarm'}
	bAlarmOutput : BOOL; //larmutgång
END_VAR
VAR
	rDevLimitInternal : REAL;
	fbDevAlarmPV: fbDevAlarm;
	rSetPointSequence1,rSetPointSequence2,rSetPointSequence3,rSetPointSequence4,rSetPointSequence5 : REAL; 	
	rTempMin,rTempMax : REAL; // tempvariabel för blockering av sekvenser 
	fbSeqLink01: Tc3_BA_Common.FB_BA_SeqLink;
	stSeqLink01 : Tc3_BA_Common.ST_BA_SeqLink;
	fbPidSeq: ARRAY[1..5] OF Tc3_BA_Common.FB_BA_SeqCtrl;
	iStartSequenceInternal : UDINT := 3;
	
	fbEdgeEnable : fbEdge;
END_VAR

fbEdgeEnable(anyInput := bEnable);
IF fbEdgeEnable.bEdgeF THEN bSync := TRUE; END_IF

fbDevAlarmPV(
	tAlarmDelay:=tAlarmDelay , 
	bAutoReset:=TRUE , 
	bAlarmOutput=>bAlarmOutput , 
	bEnable:=bEnable AND mDevAlarmCheck() , 
	rProcessValue:=rProcessValue , 
	rSetPoint:=rSetpoint , 
	rDevLimit:=rDevLimitInternal , 
	bBlockHighAlarm:=bBlockHighAlarm , 
	bBlockLowAlarm:=bBlockLowAlarm );

	IF iStartSequence > 0 AND iStartSequence < 5 THEN
	 iStartSequenceInternal	 := 5 - iStartSequence;
	END_IF;
		
IF NOT bPause THEN		
	fbSeqLink01(
	bEn:= bEnable, 
	udiSttCtrl:= iStartSequenceInternal, 
	udiIniSwiOvrDly_sec:= udiInitSwDl, 
	rX:= rProcessValue, 
	stSeqLink:=stSeqLink01 , 
	udiCurCtrl=> , 
	bSeqActv=> , 
	bNotRead=> , 
	bNoneOp=> , 
	udiRemTiIniSwiOvrDly_sec=> , 
	bErr=> , 
	sErrDescr=> );
		
	IF bBlockSequence1 THEN
		rTempMin := 0;
		rTempMax := 0;
	ELSE
		rTempMin := rMinSeq1;
		rTempMax := rMaxSeq1;
	END_IF
	rSetPointSequence1 := mCoolSetpointCheck(bActnSequence1);
	fbPidSeq[1](
	bEn:=bEnable , 
	rW:= rSetPointSequence1, 
	rX:=rProcessValue , 
	udiOpMode:= , 
	bActn:=bActnSequence1 , 
	rKp:= rKpSequence1, 
	udiTn_ms:=rKiSequence1*1000 , 
	udiTv_ms:=rDiSequence1*1000 , 
	udiTd_ms:=rFDiSequence1*1000 , 
	rYMax:=rTempMax , 
	rYMin:=rTempMin, 
	rNZ:= rDzSequence1, 
	udiCycCl:= , 
	bSync:= bSync, 
	rSync:= rSyncSeq1, 
	rYSeqInit:= rSyncSeq1, 
	udiMyNum:= 5, 
	stSeqLink:=stSeqLink01 , 
	rY=> rOutputSequence1, 
	rE=> , 
	bErr=> , 
	sErrDescr=> );
	
	IF bBlockSequence2 THEN
		rTempMin := 0;
		rTempMax := 0;
	ELSE
		rTempMin := rMinSeq2;
		rTempMax := rMaxSeq2;
	END_IF
	rSetPointSequence2 := mCoolSetpointCheck(bActnSequence2);
	fbPidSeq[2](
	bEn:=bEnable , 
	rW:= rSetPointSequence2, 
	rX:= rProcessValue, 
	udiOpMode:= , 
	bActn:= bActnSequence2, 
	rKp:= rKpSequence2, 
	udiTn_ms:=rKiSequence2*1000 , 
	udiTv_ms:=rDiSequence2*1000 , 
	udiTd_ms:=rFDiSequence2*1000 , 
	rYMax:= rTempMax, 
	rYMin:=rTempMin , 
	rNZ:= rDzSequence2, 
	udiCycCl:= , 
	bSync:= bSync, 
	rSync:= rSyncSeq2, 
	rYSeqInit:= rSyncSeq2, 
	udiMyNum:= 4, 
	stSeqLink:= stSeqLink01, 
	rY=> rOutputSequence2, 
	rE=> , 
	bErr=> , 
	sErrDescr=> );
	
	IF bBlockSequence3 THEN
		rTempMin := 0;
		rTempMax := 0;
	ELSE
		rTempMin := rMinSeq3;
		rTempMax := rMaxSeq3;
	END_IF
	rSetPointSequence3 := mCoolSetpointCheck(bActnSequence3);
	fbPidSeq[3](
	bEn:=bEnable , 
	rW:= rSetPointSequence3, 
	rX:= rProcessValue, 
	udiOpMode:= , 
	bActn:= bActnSequence3, 
	rKp:= rKpSequence3, 
	udiTn_ms:=rKiSequence3*1000 , 
	udiTv_ms:=rDiSequence3*1000 , 
	udiTd_ms:=rFDiSequence3*1000 , 
	rYMax:=rTempMax , 
	rYMin:= rTempMin, 
	rNZ:= rDzSequence3, 
	udiCycCl:= , 
	bSync:= bSync, 
	rSync:= rSyncSeq3, 
	rYSeqInit:= rSyncSeq3, 
	udiMyNum:= 3, 
	stSeqLink:= stSeqLink01, 
	rY=> rOutputSequence3, 
	rE=> , 
	bErr=> , 
	sErrDescr=> );
	
	IF bBlockSequence4 THEN
		rTempMin := 0;
		rTempMax := 0;
	ELSE
		rTempMin := rMinSeq4;
		rTempMax := rMaxSeq4;
	END_IF
	rSetPointSequence4 := mCoolSetpointCheck(bActnSequence4);
	fbPidSeq[4](
	bEn:=bEnable , 
	rW:= rSetPointSequence4, 
	rX:= rProcessValue, 
	udiOpMode:= , 
	bActn:= bActnSequence4, 
	rKp:= rKpSequence4, 
	udiTn_ms:=rKiSequence4*1000 , 
	udiTv_ms:=rDiSequence4*1000 , 
	udiTd_ms:=rFDiSequence4*1000 , 
	rYMax:=rTempMax , 
	rYMin:= rTempMin, 
	rNZ:= rDzSequence4, 
	udiCycCl:= , 
	bSync:= bSync, 
	rSync:= rSyncSeq4, 
	rYSeqInit:= rSyncSeq4, 
	udiMyNum:= 2, 
	stSeqLink:= stSeqLink01, 
	rY=> rOutputSequence4, 
	rE=> , 
	bErr=> , 
	sErrDescr=> );
	
	IF bBlockSequence5 THEN
		rTempMin := 0;
		rTempMax := 0;
	ELSE
		rTempMin := rMinSeq5;
		rTempMax := rMaxSeq5;
	END_IF
	rSetPointSequence5 := mCoolSetpointCheck(bActnSequence5);
	fbPidSeq[5](
	bEn:=bEnable , 
	rW:= rSetPointSequence5, 
	rX:= rProcessValue, 
	udiOpMode:= , 
	bActn:= bActnSequence5, 
	rKp:= rKpSequence5, 
	udiTn_ms:=rKiSequence5*1000 , 
	udiTv_ms:=rDiSequence5*1000 , 
	udiTd_ms:=rFDiSequence5*1000 , 
	rYMax:=rTempMax , 
	rYMin:= rTempMin, 
	rNZ:= rDzSequence5, 
	udiCycCl:= , 
	bSync:= bSync, 
	rSync:= rSyncSeq5, 
	rYSeqInit:= rSyncSeq5, 
	udiMyNum:= 1, 
	stSeqLink:= stSeqLink01, 
	rY=> rOutputSequence5, 
	rE=> , 
	bErr=> , 
	sErrDescr=> );
	
	bSync := FALSE;	
END_IF

IF NOT bEnable THEN
	rOutputSequence1 := rOffValSeq1;
	rOutputSequence2 := rOffValSeq2;
	rOutputSequence3 := rOffValSeq3;
	rOutputSequence4 := rOffValSeq4;
	rOutputSequence5 := rOffValSeq5;
END_IF

// Publik metod för att kolla ifall det finns någon kylsekvens i regleringen. Kan exempelvis användas för att blockera högavvikelselarm vid hög utetemperatur då kylsekvens saknas.
METHOD PUBLIC mContainsCoolingSequence : BOOL
mContainsCoolingSequence := bActnSequence1 OR bActnSequence2 OR bActnSequence3 OR bActnSequence4 OR bActnSequence5;
END_METHOD

// Metod för att kolla ifall det är en kylsekvens och om det i sådant fall är något knutet på rCoolSetpoint
METHOD PRIVATE mCoolSetpointCheck : REAL // Valt börvärde
VAR_INPUT
	bActn : BOOL; // Koll av gångriktning
END_VAR
IF NOT bActn THEN
	mCoolSetpointCheck := rSetpoint;
ELSE
	IF __ISVALIDREF(rCoolSetpoint) THEN 
		mCoolSetpointCheck := rCoolSetpoint;
	ELSE
		mCoolSetpointCheck := rSetpoint;
	END_IF
END_IF
END_METHOD

// Kolla ifall något är knutet på inputen rDevLimit. Är inget knutet där inaktiveras avvikelselarmet.
METHOD PRIVATE mDevAlarmCheck : BOOL // Valt börvärde
IF __ISVALIDREF(rDevLimit) THEN 
	mDevAlarmCheck := TRUE;
	rDevLimitInternal := rDevLimit;
ELSE
	mDevAlarmCheck := FALSE;
END_IF
END_METHOD

END_FUNCTION_BLOCK

// oaksLibrary/Regulatorer/Utökade regulatorer/fbAdvSequenceController6Stages
// Pi-regulator 6-sekvens
// För utökad kontroll av reglering:
// bPause fryser regulatorns läge
// bSync synkar regulatorns aktuella sekvens till sitt inställda rSync-värde
// udiInitSwDl är fördröjning innan byte av sekvens vid uppstart (om 0 funkar ej vald startsekvens om PV < SP)
// rSyncSeq[n] är synkvärde för resp sekvens
// rOffValSeq[n] är fast utsignal då bEnable = FALSE
{attribute 'initialize_on_call'}
FUNCTION_BLOCK fbAdvSequenceController6Stages
VAR_INPUT
	bEnable : BOOL; // Aktiverar reglering (toggla för att reset:a regulator)
	bPause : BOOL := FALSE; // Pausa regulator
	bSync : BOOL := FALSE; // Synkronisera aktuell sekvens till rSync
	udiInitSwDl : UDINT := 5; // Fördröjning för växling av sekvens vid uppstart (minst 1 om startsekvens ska gälla)	
	rProcessValue : REAL; // Aktuellt Ärvärde 
	rSetpoint : REAL; // Aktuellt börvärde. Önskas separat kylbörvärde för kylsekvenser se inputen rCoolSetpoint.
	{attribute 'initialize_on_call'}
	rCoolSetpoint : REFERENCE TO REAL; //Om man önskar ha ett högre börvärde för kylsekvenser lägg denna här så väljs detta på de sekvenser där bActnSequenceX = TRUE. Lämnar man inputen tom körs rSetpoint på både kyl och värmesekvenser.
	iStartSequence : UDINT :=3; //Sekvens där regulator startar
	
	rMinSeq1 : REAL := 0;	//Min utsignal
	rMaxSeq1 : REAL := 100;	//Max utsignal
	rSyncSeq1 : REAL := 0;	//Synkvärde
	rOffValSeq1 : REAL := 0; //Utgång om ej bEnable
	bActnSequence1 : BOOL; // Gångriktning reglersekvens  (kylsekvens = TRUE)
	bBlockSequence1 : BOOL; // blockera denna sekvens kan användas exempelvis vid nattkyla
	rKpSequence1 : REAL; // Kp
	rKiSequence1 : UDINT; // Ki
	rDiSequence1 : UDINT; // D-tid (Derivata)
	rFDiSequence1 : UDINT; // Filter tid D (Derivata)
	rDzSequence1 : REAL :=0.1; //Dödzon
	
	rMinSeq2 : REAL := 0; 
	rMaxSeq2 : REAL := 100;
	rSyncSeq2 : REAL := 0;
	rOffValSeq2 : REAL := 0; //Utgång om ej bEnable
	bActnSequence2 : BOOL; // Gångriktning reglersekvens  (kylsekvens = TRUE)
	bBlockSequence2 : BOOL; // blockera denna sekvens kan användas exempelvis vid nattkyla
	rKpSequence2 : REAL; // Kp
	rKiSequence2 : UDINT; // Ki
	rDiSequence2 : UDINT; // D-tid (Derivata)
	rFDiSequence2 : UDINT; // Filter tid D (Derivata)
	rDzSequence2 : REAL :=0.1; //Dödzon
	
	rMinSeq3 : REAL := 0; 
	rMaxSeq3 : REAL := 100;
	rSyncSeq3 : REAL := 0;
	rOffValSeq3 : REAL := 0; //Utgång om ej bEnable
	bActnSequence3 : BOOL; // Gångriktning reglersekvens  (kylsekvens = TRUE)
	bBlockSequence3 : BOOL; // blockera denna sekvens kan användas exempelvis vid nattkyla
	rKpSequence3 : REAL; // Kp
	rKiSequence3 : UDINT; // Ki
	rDiSequence3 : UDINT; // D-tid (Derivata)
	rFDiSequence3 : UDINT; // Filter tid D (Derivata)
	rDzSequence3 : REAL :=0.1; //Dödzon
	
	rMinSeq4 : REAL := 0; 
	rMaxSeq4 : REAL := 100;
	rSyncSeq4 : REAL := 0;
	rOffValSeq4 : REAL := 0; //Utgång om ej bEnable
	bActnSequence4 : BOOL; // Gångriktning reglersekvens  (kylsekvens = TRUE)
	bBlockSequence4 : BOOL; // blockera denna sekvens kan användas exempelvis vid nattkyla
	rKpSequence4 : REAL; // Kp
	rKiSequence4 : UDINT; // Ki
	rDiSequence4 : UDINT; // D-tid (Derivata)
	rFDiSequence4 : UDINT; // Filter tid D (Derivata)
	rDzSequence4 : REAL :=0.1; //Dödzon
	
	rMinSeq5 : REAL := 0; 
	rMaxSeq5 : REAL := 100;
	rSyncSeq5 : REAL := 0;
	rOffValSeq5 : REAL := 0; //Utgång om ej bEnable
	bActnSequence5 : BOOL; // Gångriktning reglersekvens  (kylsekvens = TRUE)
	bBlockSequence5 : BOOL; // blockera denna sekvens kan användas exempelvis vid nattkyla
	rKpSequence5 : REAL; // Kp
	rKiSequence5 : UDINT; // Ki
	rDiSequence5 : UDINT; // D-tid (Derivata)
	rFDiSequence5 : UDINT; // Filter tid D (Derivata)
	rDzSequence5 : REAL :=0.1; //Dödzon
	
	rMinSeq6 : REAL := 0; 
	rMaxSeq6 : REAL := 100;
	rSyncSeq6 : REAL := 0;
	rOffValSeq6 : REAL := 0; //Utgång om ej bEnable
	bActnSequence6 : BOOL; // Gångriktning reglersekvens  (kylsekvens = TRUE)
	bBlockSequence6 : BOOL; // blockera denna sekvens kan användas exempelvis vid nattkyla
	rKpSequence6 : REAL; // Kp
	rKiSequence6 : UDINT; // Ki
	rDiSequence6 : UDINT; // D-tid (Derivata)
	rFDiSequence6 : UDINT; // Filter tid D (Derivata)
	rDzSequence6 : REAL :=0.1; //Dödzon
	
	{attribute 'pingroup' := 'DeviationAlarm'}
	{attribute 'initialize_on_call'}
	rDevLimit : REFERENCE TO REAL := 0;
	{attribute 'pingroup' := 'DeviationAlarm'}
	bBlockHighAlarm : BOOL; // Blockera högtemplarm
	{attribute 'pingroup' := 'DeviationAlarm'}
	bBlockLowAlarm : BOOL; // Blockera lågtemplarm
	{attribute 'pingroup' := 'DeviationAlarm'}
	tAlarmDelay : TIME := T#5S; // larmfördröjning
END_VAR
VAR_OUTPUT
	rY : REAL; // Utsignal huvudregulator
	rOutputSequence1 : REAL;  // regulatorsignal
	rOutputSequence2 : REAL;  // regulatorsignal
	rOutputSequence3 : REAL;  // regulatorsignal
	rOutputSequence4 : REAL;  // regulatorsignal
	rOutputSequence5 : REAL;  // regulatorsignal
	rOutputSequence6 : REAL;  // regulatorsignal
	{attribute 'pingroup' := 'DeviationAlarm'}
	bAlarmOutput : BOOL; //larmutgång
END_VAR
VAR
	rDevLimitInternal : REAL;
	fbDevAlarmPV: fbDevAlarm;
	rSetPointSequence1,rSetPointSequence2,rSetPointSequence3,rSetPointSequence4,rSetPointSequence5,rSetPointSequence6 : REAL; 	
	rTempMin,rTempMax : REAL; // tempvariabel för blockering av sekvenser 
	fbSeqLink01: Tc3_BA_Common.FB_BA_SeqLink;
	stSeqLink01 : Tc3_BA_Common.ST_BA_SeqLink;
	fbPidSeq: ARRAY[1..6] OF Tc3_BA_Common.FB_BA_SeqCtrl;
	iStartSequenceInternal : UDINT := 3;
	
	fbEdgeEnable : fbEdge;
END_VAR

fbEdgeEnable(anyInput := bEnable);
IF fbEdgeEnable.bEdgeF THEN bSync := TRUE; END_IF

fbDevAlarmPV(
	tAlarmDelay:=tAlarmDelay , 
	bAutoReset:=TRUE , 
	bAlarmOutput=>bAlarmOutput , 
	bEnable:=bEnable AND mDevAlarmCheck() , 
	rProcessValue:=rProcessValue , 
	rSetPoint:=rSetpoint , 
	rDevLimit:=rDevLimitInternal , 
	bBlockHighAlarm:=bBlockHighAlarm , 
	bBlockLowAlarm:=bBlockLowAlarm );

	IF iStartSequence > 0 AND iStartSequence < 6 THEN
	 iStartSequenceInternal	 := 6 - iStartSequence;
	END_IF;
		
IF NOT bPause THEN		
	fbSeqLink01(
	bEn:= bEnable, 
	udiSttCtrl:= iStartSequenceInternal, 
	udiIniSwiOvrDly_sec:= udiInitSwDl, 
	rX:= rProcessValue, 
	stSeqLink:=stSeqLink01 , 
	udiCurCtrl=> , 
	bSeqActv=> , 
	bNotRead=> , 
	bNoneOp=> , 
	udiRemTiIniSwiOvrDly_sec=> , 
	bErr=> , 
	sErrDescr=> );
		
	IF bBlockSequence1 THEN
		rTempMin := 0;
		rTempMax := 0;
	ELSE
		rTempMin := rMinSeq1;
		rTempMax := rMaxSeq1;
	END_IF
	rSetPointSequence1 := mCoolSetpointCheck(bActnSequence1);
	fbPidSeq[1](
	bEn:=bEnable , 
	rW:= rSetPointSequence1, 
	rX:=rProcessValue , 
	udiOpMode:= , 
	bActn:=bActnSequence1 , 
	rKp:= rKpSequence1, 
	udiTn_ms:=rKiSequence1*1000 , 
	udiTv_ms:=rDiSequence1*1000 , 
	udiTd_ms:=rFDiSequence1*1000 , 
	rYMax:=rTempMax , 
	rYMin:=rTempMin, 
	rNZ:= rDzSequence1, 
	udiCycCl:= , 
	bSync:= bSync, 
	rSync:= rSyncSeq1, 
	rYSeqInit:= rSyncSeq1, 
	udiMyNum:= 6, 
	stSeqLink:=stSeqLink01 , 
	rY=> rOutputSequence1, 
	rE=> , 
	bErr=> , 
	sErrDescr=> );
	
	IF bBlockSequence2 THEN
		rTempMin := 0;
		rTempMax := 0;
	ELSE
		rTempMin := rMinSeq2;
		rTempMax := rMaxSeq2;
	END_IF
	rSetPointSequence2 := mCoolSetpointCheck(bActnSequence2);
	fbPidSeq[2](
	bEn:=bEnable , 
	rW:= rSetPointSequence2, 
	rX:= rProcessValue, 
	udiOpMode:= , 
	bActn:= bActnSequence2, 
	rKp:= rKpSequence2, 
	udiTn_ms:=rKiSequence2*1000 , 
	udiTv_ms:=rDiSequence2*1000 , 
	udiTd_ms:=rFDiSequence2*1000 , 
	rYMax:= rTempMax, 
	rYMin:=rTempMin , 
	rNZ:= rDzSequence2, 
	udiCycCl:= , 
	bSync:= bSync, 
	rSync:= rSyncSeq2, 
	rYSeqInit:= rSyncSeq2, 
	udiMyNum:= 5, 
	stSeqLink:= stSeqLink01, 
	rY=> rOutputSequence2, 
	rE=> , 
	bErr=> , 
	sErrDescr=> );
	
	IF bBlockSequence3 THEN
		rTempMin := 0;
		rTempMax := 0;
	ELSE
		rTempMin := rMinSeq3;
		rTempMax := rMaxSeq3;
	END_IF
	rSetPointSequence3 := mCoolSetpointCheck(bActnSequence3);
	fbPidSeq[3](
	bEn:=bEnable , 
	rW:= rSetPointSequence3, 
	rX:= rProcessValue, 
	udiOpMode:= , 
	bActn:= bActnSequence3, 
	rKp:= rKpSequence3, 
	udiTn_ms:=rKiSequence3*1000 , 
	udiTv_ms:=rDiSequence3*1000 , 
	udiTd_ms:=rFDiSequence3*1000 , 
	rYMax:=rTempMax , 
	rYMin:= rTempMin, 
	rNZ:= rDzSequence3, 
	udiCycCl:= , 
	bSync:= bSync, 
	rSync:= rSyncSeq3, 
	rYSeqInit:= rSyncSeq3, 
	udiMyNum:= 4, 
	stSeqLink:= stSeqLink01, 
	rY=> rOutputSequence3, 
	rE=> , 
	bErr=> , 
	sErrDescr=> );
	
	IF bBlockSequence4 THEN
		rTempMin := 0;
		rTempMax := 0;
	ELSE
		rTempMin := rMinSeq4;
		rTempMax := rMaxSeq4;
	END_IF
	rSetPointSequence4 := mCoolSetpointCheck(bActnSequence4);
	fbPidSeq[4](
	bEn:=bEnable , 
	rW:= rSetPointSequence4, 
	rX:= rProcessValue, 
	udiOpMode:= , 
	bActn:= bActnSequence4, 
	rKp:= rKpSequence4, 
	udiTn_ms:=rKiSequence4*1000 , 
	udiTv_ms:=rDiSequence4*1000 , 
	udiTd_ms:=rFDiSequence4*1000 , 
	rYMax:=rTempMax , 
	rYMin:= rTempMin, 
	rNZ:= rDzSequence4, 
	udiCycCl:= , 
	bSync:= bSync, 
	rSync:= rSyncSeq4, 
	rYSeqInit:= rSyncSeq4, 
	udiMyNum:= 3, 
	stSeqLink:= stSeqLink01, 
	rY=> rOutputSequence4, 
	rE=> , 
	bErr=> , 
	sErrDescr=> );
	
	IF bBlockSequence5 THEN
		rTempMin := 0;
		rTempMax := 0;
	ELSE
		rTempMin := rMinSeq5;
		rTempMax := rMaxSeq5;
	END_IF
	rSetPointSequence5 := mCoolSetpointCheck(bActnSequence5);
	fbPidSeq[5](
	bEn:=bEnable , 
	rW:= rSetPointSequence5, 
	rX:= rProcessValue, 
	udiOpMode:= , 
	bActn:= bActnSequence5, 
	rKp:= rKpSequence5, 
	udiTn_ms:=rKiSequence5*1000 , 
	udiTv_ms:=rDiSequence5*1000 , 
	udiTd_ms:=rFDiSequence5*1000 , 
	rYMax:=rTempMax , 
	rYMin:= rTempMin, 
	rNZ:= rDzSequence5, 
	udiCycCl:= , 
	bSync:= bSync, 
	rSync:= rSyncSeq5, 
	rYSeqInit:= rSyncSeq5, 
	udiMyNum:= 2, 
	stSeqLink:= stSeqLink01, 
	rY=> rOutputSequence5, 
	rE=> , 
	bErr=> , 
	sErrDescr=> );
	
	IF bBlockSequence6 THEN
		rTempMin := 0;
		rTempMax := 0;
	ELSE
		rTempMin := rMinSeq6;
		rTempMax := rMaxSeq6;
	END_IF
	rSetPointSequence6 := mCoolSetpointCheck(bActnSequence6);
	fbPidSeq[6](
	bEn:=bEnable , 
	rW:= rSetPointSequence6, 
	rX:= rProcessValue, 
	udiOpMode:= , 
	bActn:= bActnSequence6, 
	rKp:= rKpSequence6, 
	udiTn_ms:=rKiSequence6*1000 , 
	udiTv_ms:=rDiSequence6*1000 , 
	udiTd_ms:=rFDiSequence6*1000 , 
	rYMax:=rTempMax , 
	rYMin:= rTempMin, 
	rNZ:= rDzSequence6, 
	udiCycCl:= , 
	bSync:= bSync, 
	rSync:= rSyncSeq6, 
	rYSeqInit:= rSyncSeq6, 
	udiMyNum:= 1, 
	stSeqLink:= stSeqLink01, 
	rY=> rOutputSequence6, 
	rE=> , 
	bErr=> , 
	sErrDescr=> );
	
	bSync := FALSE;	
END_IF

IF NOT bEnable THEN
	rOutputSequence1 := rOffValSeq1;
	rOutputSequence2 := rOffValSeq2;
	rOutputSequence3 := rOffValSeq3;
	rOutputSequence4 := rOffValSeq4;
	rOutputSequence5 := rOffValSeq5;
	rOutputSequence6 := rOffValSeq6;
END_IF

// Publik metod för att kolla ifall det finns någon kylsekvens i regleringen. Kan exempelvis användas för att blockera högavvikelselarm vid hög utetemperatur då kylsekvens saknas.
METHOD PUBLIC mContainsCoolingSequence : BOOL
mContainsCoolingSequence := bActnSequence1 OR bActnSequence2 OR bActnSequence3 OR bActnSequence4 OR bActnSequence5;
END_METHOD

// Metod för att kolla ifall det är en kylsekvens och om det i sådant fall är något knutet på rCoolSetpoint
METHOD PRIVATE mCoolSetpointCheck : REAL // Valt börvärde
VAR_INPUT
	bActn : BOOL; // Koll av gångriktning
END_VAR
IF NOT bActn THEN
	mCoolSetpointCheck := rSetpoint;
ELSE
	IF __ISVALIDREF(rCoolSetpoint) THEN 
		mCoolSetpointCheck := rCoolSetpoint;
	ELSE
		mCoolSetpointCheck := rSetpoint;
	END_IF
END_IF
END_METHOD

// Kolla ifall något är knutet på inputen rDevLimit. Är inget knutet där inaktiveras avvikelselarmet.
METHOD PRIVATE mDevAlarmCheck : BOOL // Valt börvärde
IF __ISVALIDREF(rDevLimit) THEN 
	mDevAlarmCheck := TRUE;
	rDevLimitInternal := rDevLimit;
ELSE
	mDevAlarmCheck := FALSE;
END_IF
END_METHOD

END_FUNCTION_BLOCK

// oaksLibrary/Regulatorer/Utökade regulatorer/fbAdvSequenceController7Stages
// Pi-regulator 7-sekvens
// För utökad kontroll av reglering:
// bPause fryser regulatorns läge
// bSync synkar regulatorns aktuella sekvens till sitt inställda rSync-värde
// udiInitSwDl är fördröjning innan byte av sekvens vid uppstart (om 0 funkar ej vald startsekvens om PV < SP)
// rSyncSeq[n] är synkvärde för resp sekvens
// rOffValSeq[n] är fast utsignal då bEnable = FALSE
{attribute 'initialize_on_call'}
FUNCTION_BLOCK fbAdvSequenceController7Stages
VAR_INPUT
	bEnable : BOOL; // Aktiverar reglering (toggla för att reset:a regulator)
	bPause : BOOL := FALSE; // Pausa regulator
	bSync : BOOL := FALSE; // Synkronisera aktuell sekvens till rSync
	udiInitSwDl : UDINT := 5; // Fördröjning för växling av sekvens vid uppstart (minst 1 om startsekvens ska gälla)	
	rProcessValue : REAL; // Aktuellt Ärvärde 
	rSetpoint : REAL; // Aktuellt börvärde. Önskas separat kylbörvärde för kylsekvenser se inputen rCoolSetpoint.
	{attribute 'initialize_on_call'}
	rCoolSetpoint : REFERENCE TO REAL; //Om man önskar ha ett högre börvärde för kylsekvenser lägg denna här så väljs detta på de sekvenser där bActnSequenceX = TRUE. Lämnar man inputen tom körs rSetpoint på både kyl och värmesekvenser.
	iStartSequence : UDINT :=3; //Sekvens där regulator startar
	
	rMinSeq1 : REAL := 0;	//Min utsignal
	rMaxSeq1 : REAL := 100;	//Max utsignal
	rSyncSeq1 : REAL := 0;	//Synkvärde
	rOffValSeq1 : REAL := 0; //Utgång om ej bEnable
	bActnSequence1 : BOOL; // Gångriktning reglersekvens  (kylsekvens = TRUE)
	bBlockSequence1 : BOOL; // blockera denna sekvens kan användas exempelvis vid nattkyla
	rKpSequence1 : REAL; // Kp
	rKiSequence1 : UDINT; // Ki
	rDiSequence1 : UDINT; // D-tid (Derivata)
	rFDiSequence1 : UDINT; // Filter tid D (Derivata)
	rDzSequence1 : REAL :=0.1; //Dödzon
	
	rMinSeq2 : REAL := 0; 
	rMaxSeq2 : REAL := 100;
	rSyncSeq2 : REAL := 0;
	rOffValSeq2 : REAL := 0; //Utgång om ej bEnable
	bActnSequence2 : BOOL; // Gångriktning reglersekvens  (kylsekvens = TRUE)
	bBlockSequence2 : BOOL; // blockera denna sekvens kan användas exempelvis vid nattkyla
	rKpSequence2 : REAL; // Kp
	rKiSequence2 : UDINT; // Ki
	rDiSequence2 : UDINT; // D-tid (Derivata)
	rFDiSequence2 : UDINT; // Filter tid D (Derivata)
	rDzSequence2 : REAL :=0.1; //Dödzon
	
	rMinSeq3 : REAL := 0; 
	rMaxSeq3 : REAL := 100;
	rSyncSeq3 : REAL := 0;
	rOffValSeq3 : REAL := 0; //Utgång om ej bEnable
	bActnSequence3 : BOOL; // Gångriktning reglersekvens  (kylsekvens = TRUE)
	bBlockSequence3 : BOOL; // blockera denna sekvens kan användas exempelvis vid nattkyla
	rKpSequence3 : REAL; // Kp
	rKiSequence3 : UDINT; // Ki
	rDiSequence3 : UDINT; // D-tid (Derivata)
	rFDiSequence3 : UDINT; // Filter tid D (Derivata)
	rDzSequence3 : REAL :=0.1; //Dödzon
	
	rMinSeq4 : REAL := 0; 
	rMaxSeq4 : REAL := 100;
	rSyncSeq4 : REAL := 0;
	rOffValSeq4 : REAL := 0; //Utgång om ej bEnable
	bActnSequence4 : BOOL; // Gångriktning reglersekvens  (kylsekvens = TRUE)
	bBlockSequence4 : BOOL; // blockera denna sekvens kan användas exempelvis vid nattkyla
	rKpSequence4 : REAL; // Kp
	rKiSequence4 : UDINT; // Ki
	rDiSequence4 : UDINT; // D-tid (Derivata)
	rFDiSequence4 : UDINT; // Filter tid D (Derivata)
	rDzSequence4 : REAL :=0.1; //Dödzon
	
	rMinSeq5 : REAL := 0; 
	rMaxSeq5 : REAL := 100;
	rSyncSeq5 : REAL := 0;
	rOffValSeq5 : REAL := 0; //Utgång om ej bEnable
	bActnSequence5 : BOOL; // Gångriktning reglersekvens  (kylsekvens = TRUE)
	bBlockSequence5 : BOOL; // blockera denna sekvens kan användas exempelvis vid nattkyla
	rKpSequence5 : REAL; // Kp
	rKiSequence5 : UDINT; // Ki
	rDiSequence5 : UDINT; // D-tid (Derivata)
	rFDiSequence5 : UDINT; // Filter tid D (Derivata)
	rDzSequence5 : REAL :=0.1; //Dödzon
	
	rMinSeq6 : REAL := 0; 
	rMaxSeq6 : REAL := 100;
	rSyncSeq6 : REAL := 0;
	rOffValSeq6 : REAL := 0; //Utgång om ej bEnable
	bActnSequence6 : BOOL; // Gångriktning reglersekvens  (kylsekvens = TRUE)
	bBlockSequence6 : BOOL; // blockera denna sekvens kan användas exempelvis vid nattkyla
	rKpSequence6 : REAL; // Kp
	rKiSequence6 : UDINT; // Ki
	rDiSequence6 : UDINT; // D-tid (Derivata)
	rFDiSequence6 : UDINT; // Filter tid D (Derivata)
	rDzSequence6 : REAL :=0.1; //Dödzon
	
	rMinSeq7 : REAL := 0; 
	rMaxSeq7 : REAL := 100;
	rSyncSeq7 : REAL := 0;
	rOffValSeq7 : REAL := 0; //Utgång om ej bEnable
	bActnSequence7 : BOOL; // Gångriktning reglersekvens  (kylsekvens = TRUE)
	bBlockSequence7 : BOOL; // blockera denna sekvens kan användas exempelvis vid nattkyla
	rKpSequence7 : REAL; // Kp
	rKiSequence7 : UDINT; // Ki
	rDiSequence7 : UDINT; // D-tid (Derivata)
	rFDiSequence7 : UDINT; // Filter tid D (Derivata)
	rDzSequence7 : REAL :=0.1; //Dödzon
	
	{attribute 'pingroup' := 'DeviationAlarm'}
	{attribute 'initialize_on_call'}
	rDevLimit : REFERENCE TO REAL := 0;
	{attribute 'pingroup' := 'DeviationAlarm'}
	bBlockHighAlarm : BOOL; // Blockera högtemplarm
	{attribute 'pingroup' := 'DeviationAlarm'}
	bBlockLowAlarm : BOOL; // Blockera lågtemplarm
	{attribute 'pingroup' := 'DeviationAlarm'}
	tAlarmDelay : TIME := T#5S; // larmfördröjning
END_VAR
VAR_OUTPUT
	rY : REAL; // Utsignal huvudregulator
	rOutputSequence1 : REAL;  // regulatorsignal
	rOutputSequence2 : REAL;  // regulatorsignal
	rOutputSequence3 : REAL;  // regulatorsignal
	rOutputSequence4 : REAL;  // regulatorsignal
	rOutputSequence5 : REAL;  // regulatorsignal
	rOutputSequence6 : REAL;  // regulatorsignal
	rOutputSequence7 : REAL;  // regulatorsignal
	{attribute 'pingroup' := 'DeviationAlarm'}
	bAlarmOutput : BOOL; //larmutgång
END_VAR
VAR
	rDevLimitInternal : REAL;
	fbDevAlarmPV: fbDevAlarm;
	rSetPointSequence1,rSetPointSequence2,rSetPointSequence3,rSetPointSequence4,rSetPointSequence5,rSetPointSequence6,rSetPointSequence7 : REAL; 	
	rTempMin,rTempMax : REAL; // tempvariabel för blockering av sekvenser 
	fbSeqLink01: Tc3_BA_Common.FB_BA_SeqLink;
	stSeqLink01 : Tc3_BA_Common.ST_BA_SeqLink;
	fbPidSeq: ARRAY[1..7] OF Tc3_BA_Common.FB_BA_SeqCtrl;
	iStartSequenceInternal : UDINT := 3;
	
	fbEdgeEnable : fbEdge;
END_VAR

fbEdgeEnable(anyInput := bEnable);
IF fbEdgeEnable.bEdgeF THEN bSync := TRUE; END_IF

fbDevAlarmPV(
	tAlarmDelay:=tAlarmDelay , 
	bAutoReset:=TRUE , 
	bAlarmOutput=>bAlarmOutput , 
	bEnable:=bEnable AND mDevAlarmCheck() , 
	rProcessValue:=rProcessValue , 
	rSetPoint:=rSetpoint , 
	rDevLimit:=rDevLimitInternal , 
	bBlockHighAlarm:=bBlockHighAlarm , 
	bBlockLowAlarm:=bBlockLowAlarm );

	IF iStartSequence > 0 AND iStartSequence < 7 THEN
	 iStartSequenceInternal	 := 7 - iStartSequence;
	END_IF;
		
IF NOT bPause THEN		
	fbSeqLink01(
	bEn:= bEnable, 
	udiSttCtrl:= iStartSequenceInternal, 
	udiIniSwiOvrDly_sec:= udiInitSwDl, 
	rX:= rProcessValue, 
	stSeqLink:=stSeqLink01 , 
	udiCurCtrl=> , 
	bSeqActv=> , 
	bNotRead=> , 
	bNoneOp=> , 
	udiRemTiIniSwiOvrDly_sec=> , 
	bErr=> , 
	sErrDescr=> );
		
	IF bBlockSequence1 THEN
		rTempMin := 0;
		rTempMax := 0;
	ELSE
		rTempMin := rMinSeq1;
		rTempMax := rMaxSeq1;
	END_IF
	rSetPointSequence1 := mCoolSetpointCheck(bActnSequence1);
	fbPidSeq[1](
	bEn:=bEnable , 
	rW:= rSetPointSequence1, 
	rX:=rProcessValue , 
	udiOpMode:= , 
	bActn:=bActnSequence1 , 
	rKp:= rKpSequence1, 
	udiTn_ms:=rKiSequence1*1000 , 
	udiTv_ms:=rDiSequence1*1000 , 
	udiTd_ms:=rFDiSequence1*1000 , 
	rYMax:=rTempMax , 
	rYMin:=rTempMin, 
	rNZ:= rDzSequence1, 
	udiCycCl:= , 
	bSync:= bSync, 
	rSync:= rSyncSeq1, 
	rYSeqInit:= rSyncSeq1, 
	udiMyNum:= 7, 
	stSeqLink:=stSeqLink01 , 
	rY=> rOutputSequence1, 
	rE=> , 
	bErr=> , 
	sErrDescr=> );
	
	IF bBlockSequence2 THEN
		rTempMin := 0;
		rTempMax := 0;
	ELSE
		rTempMin := rMinSeq2;
		rTempMax := rMaxSeq2;
	END_IF
	rSetPointSequence2 := mCoolSetpointCheck(bActnSequence2);
	fbPidSeq[2](
	bEn:=bEnable , 
	rW:= rSetPointSequence2, 
	rX:= rProcessValue, 
	udiOpMode:= , 
	bActn:= bActnSequence2, 
	rKp:= rKpSequence2, 
	udiTn_ms:=rKiSequence2*1000 , 
	udiTv_ms:=rDiSequence2*1000 , 
	udiTd_ms:=rFDiSequence2*1000 , 
	rYMax:= rTempMax, 
	rYMin:=rTempMin , 
	rNZ:= rDzSequence2, 
	udiCycCl:= , 
	bSync:= bSync, 
	rSync:= rSyncSeq2, 
	rYSeqInit:= rSyncSeq2, 
	udiMyNum:= 6, 
	stSeqLink:= stSeqLink01, 
	rY=> rOutputSequence2, 
	rE=> , 
	bErr=> , 
	sErrDescr=> );
	
	IF bBlockSequence3 THEN
		rTempMin := 0;
		rTempMax := 0;
	ELSE
		rTempMin := rMinSeq3;
		rTempMax := rMaxSeq3;
	END_IF
	rSetPointSequence3 := mCoolSetpointCheck(bActnSequence3);
	fbPidSeq[3](
	bEn:=bEnable , 
	rW:= rSetPointSequence3, 
	rX:= rProcessValue, 
	udiOpMode:= , 
	bActn:= bActnSequence3, 
	rKp:= rKpSequence3, 
	udiTn_ms:=rKiSequence3*1000 , 
	udiTv_ms:=rDiSequence3*1000 , 
	udiTd_ms:=rFDiSequence3*1000 , 
	rYMax:=rTempMax , 
	rYMin:= rTempMin, 
	rNZ:= rDzSequence3, 
	udiCycCl:= , 
	bSync:= bSync, 
	rSync:= rSyncSeq3, 
	rYSeqInit:= rSyncSeq3, 
	udiMyNum:= 5, 
	stSeqLink:= stSeqLink01, 
	rY=> rOutputSequence3, 
	rE=> , 
	bErr=> , 
	sErrDescr=> );
	
	IF bBlockSequence4 THEN
		rTempMin := 0;
		rTempMax := 0;
	ELSE
		rTempMin := rMinSeq4;
		rTempMax := rMaxSeq4;
	END_IF
	rSetPointSequence4 := mCoolSetpointCheck(bActnSequence4);
	fbPidSeq[4](
	bEn:=bEnable , 
	rW:= rSetPointSequence4, 
	rX:= rProcessValue, 
	udiOpMode:= , 
	bActn:= bActnSequence4, 
	rKp:= rKpSequence4, 
	udiTn_ms:=rKiSequence4*1000 , 
	udiTv_ms:=rDiSequence4*1000 , 
	udiTd_ms:=rFDiSequence4*1000 , 
	rYMax:=rTempMax , 
	rYMin:= rTempMin, 
	rNZ:= rDzSequence4, 
	udiCycCl:= , 
	bSync:= bSync, 
	rSync:= rSyncSeq4, 
	rYSeqInit:= rSyncSeq4, 
	udiMyNum:= 4, 
	stSeqLink:= stSeqLink01, 
	rY=> rOutputSequence4, 
	rE=> , 
	bErr=> , 
	sErrDescr=> );
	
	IF bBlockSequence5 THEN
		rTempMin := 0;
		rTempMax := 0;
	ELSE
		rTempMin := rMinSeq5;
		rTempMax := rMaxSeq5;
	END_IF
	rSetPointSequence5 := mCoolSetpointCheck(bActnSequence5);
	fbPidSeq[5](
	bEn:=bEnable , 
	rW:= rSetPointSequence5, 
	rX:= rProcessValue, 
	udiOpMode:= , 
	bActn:= bActnSequence5, 
	rKp:= rKpSequence5, 
	udiTn_ms:=rKiSequence5*1000 , 
	udiTv_ms:=rDiSequence5*1000 , 
	udiTd_ms:=rFDiSequence5*1000 , 
	rYMax:=rTempMax , 
	rYMin:= rTempMin, 
	rNZ:= rDzSequence5, 
	udiCycCl:= , 
	bSync:= bSync, 
	rSync:= rSyncSeq5, 
	rYSeqInit:= rSyncSeq5, 
	udiMyNum:= 3, 
	stSeqLink:= stSeqLink01, 
	rY=> rOutputSequence5, 
	rE=> , 
	bErr=> , 
	sErrDescr=> );
	
	IF bBlockSequence6 THEN
		rTempMin := 0;
		rTempMax := 0;
	ELSE
		rTempMin := rMinSeq6;
		rTempMax := rMaxSeq6;
	END_IF
	rSetPointSequence6 := mCoolSetpointCheck(bActnSequence6);
	fbPidSeq[6](
	bEn:=bEnable , 
	rW:= rSetPointSequence6, 
	rX:= rProcessValue, 
	udiOpMode:= , 
	bActn:= bActnSequence6, 
	rKp:= rKpSequence6, 
	udiTn_ms:=rKiSequence6*1000 , 
	udiTv_ms:=rDiSequence6*1000 , 
	udiTd_ms:=rFDiSequence6*1000 , 
	rYMax:=rTempMax , 
	rYMin:= rTempMin, 
	rNZ:= rDzSequence6, 
	udiCycCl:= , 
	bSync:= bSync, 
	rSync:= rSyncSeq6, 
	rYSeqInit:= rSyncSeq6, 
	udiMyNum:= 2, 
	stSeqLink:= stSeqLink01, 
	rY=> rOutputSequence6, 
	rE=> , 
	bErr=> , 
	sErrDescr=> );
	
	IF bBlockSequence7 THEN
		rTempMin := 0;
		rTempMax := 0;
	ELSE
		rTempMin := rMinSeq7;
		rTempMax := rMaxSeq7;
	END_IF
	rSetPointSequence7 := mCoolSetpointCheck(bActnSequence7);
	fbPidSeq[7](
	bEn:=bEnable , 
	rW:= rSetPointSequence7, 
	rX:= rProcessValue, 
	udiOpMode:= , 
	bActn:= bActnSequence7, 
	rKp:= rKpSequence7, 
	udiTn_ms:=rKiSequence7*1000 , 
	udiTv_ms:=rDiSequence7*1000 , 
	udiTd_ms:=rFDiSequence7*1000 , 
	rYMax:=rTempMax , 
	rYMin:= rTempMin, 
	rNZ:= rDzSequence7, 
	udiCycCl:= , 
	bSync:= bSync, 
	rSync:= rSyncSeq7, 
	rYSeqInit:= rSyncSeq7, 
	udiMyNum:= 1, 
	stSeqLink:= stSeqLink01, 
	rY=> rOutputSequence7, 
	rE=> , 
	bErr=> , 
	sErrDescr=> );
	
	bSync := FALSE;	
END_IF

IF NOT bEnable THEN
	rOutputSequence1 := rOffValSeq1;
	rOutputSequence2 := rOffValSeq2;
	rOutputSequence3 := rOffValSeq3;
	rOutputSequence4 := rOffValSeq4;
	rOutputSequence5 := rOffValSeq5;
	rOutputSequence6 := rOffValSeq6;
	rOutputSequence7 := rOffValSeq7;
END_IF

// Publik metod för att kolla ifall det finns någon kylsekvens i regleringen. Kan exempelvis användas för att blockera högavvikelselarm vid hög utetemperatur då kylsekvens saknas.
METHOD PUBLIC mContainsCoolingSequence : BOOL
mContainsCoolingSequence := bActnSequence1 OR bActnSequence2 OR bActnSequence3 OR bActnSequence4 OR bActnSequence5;
END_METHOD

// Metod för att kolla ifall det är en kylsekvens och om det i sådant fall är något knutet på rCoolSetpoint
METHOD PRIVATE mCoolSetpointCheck : REAL // Valt börvärde
VAR_INPUT
	bActn : BOOL; // Koll av gångriktning
END_VAR
IF NOT bActn THEN
	mCoolSetpointCheck := rSetpoint;
ELSE
	IF __ISVALIDREF(rCoolSetpoint) THEN 
		mCoolSetpointCheck := rCoolSetpoint;
	ELSE
		mCoolSetpointCheck := rSetpoint;
	END_IF
END_IF
END_METHOD

// Kolla ifall något är knutet på inputen rDevLimit. Är inget knutet där inaktiveras avvikelselarmet.
METHOD PRIVATE mDevAlarmCheck : BOOL // Valt börvärde
IF __ISVALIDREF(rDevLimit) THEN 
	mDevAlarmCheck := TRUE;
	rDevLimitInternal := rDevLimit;
ELSE
	mDevAlarmCheck := FALSE;
END_IF
END_METHOD

END_FUNCTION_BLOCK

// oaksLibrary/Regulatorer/fbSequenceController2Stages
// Pi-regulator 2-sekvens
{attribute 'initialize_on_call'}
FUNCTION_BLOCK fbSequenceController2Stages
VAR_INPUT
	bEnable : BOOL; // Aktiverar reglering
	rProcessValue : REAL; // Aktuellt Ärvärde 
	rSetpoint : REAL; // Aktuellt börvärde. Önskas separat kylbörvärde för kylsekvenser se inputen rCoolSetpoint.
	{attribute 'initialize_on_call'}
	rCoolSetpoint : REFERENCE TO REAL := 0; //Om man önskar ha ett högre börvärde för kylsekvenser lägg denna här så väljs detta på de sekvenser där bActnSequenceX = TRUE. Lämnar man inputen tom körs rSetpoint på både kyl och värmesekvenser.
	rMinSeq1 : REAL := 0; 
	rMaxSeq1 : REAL := 100; 
	bActnSequence1 : BOOL; // Gångriktning reglersekvens  (kylsekvens = TRUE)
	bBlockSequence1 : BOOL; // blockera denna sekvens kan användas exempelvis vid nattkyla
	rMinSeq2 : REAL := 0; 
	rMaxSeq2 : REAL := 100; 
	bActnSequence2 : BOOL; // Gångriktning reglersekvens  (kylsekvens = TRUE)
	bBlockSequence2 : BOOL; // blockera denna sekvens kan användas exempelvis vid nattkyla
	rKpSequence1 : REAL; // Kp
	rKiSequence1 : UDINT; // Ki
	rDiSequence1 : UDINT; // D-tid (Derivata)
	rFDiSequence1 : UDINT; // Filter tid D (Derivata)
	rDzSequence1 : REAL :=0.1; //Dödzon
	rKpSequence2 : REAL; // Kp
	rKiSequence2 : UDINT; // Ki
	rDiSequence2 : UDINT; // D-tid (Derivata)
	rFDiSequence2 : UDINT; // Filter tid D (Derivata)
	rDzSequence2 : REAL :=0.1; //Dödzon
	iStartSequence : UDINT :=2; //Sekvens där regulator startar
	{attribute 'initialize_on_call'}
	rDevLimit : REFERENCE TO REAL := 0;
	{attribute 'pingroup' := 'DeviationAlarm'}
	bBlockHighAlarm : BOOL; // Blockera högtemplarm
	{attribute 'pingroup' := 'DeviationAlarm'}
	bBlockLowAlarm : BOOL; // Blockera lågtemplarm
	{attribute 'pingroup' := 'DeviationAlarm'}
	tAlarmDelay : TIME := T#5S; // larmfördröjning
END_VAR
VAR_OUTPUT
	rOutputSequence1 : REAL;  // regulatorsignal
	rOutputSequence2 : REAL;  // regulatorsignal
	{attribute 'pingroup' := 'DeviationAlarm'}
	bAlarmOutput : BOOL; //larmutgång
END_VAR
VAR
	rDevLimitInternal : REAL;
	fbDevAlarmPV: fbDevAlarm;
	rSetPointSequence1,rSetPointSequence2 : REAL; 	

	rTempMin,rTempMax : REAL; // tempvariabel för blockering av sekvenser 
	fbSeqLink01: Tc3_BA_Common.FB_BA_SeqLink;
	stSeqLink01 : Tc3_BA_Common.ST_BA_SeqLink;
	fbPidSeq: ARRAY[1..2] OF Tc3_BA_Common.FB_BA_SeqCtrl;
	iStartSequenceInternal : UDINT := 2;
END_VAR

	fbDevAlarmPV(
	tAlarmDelay:=tAlarmDelay , 
	bAutoReset:=TRUE , 
	bAlarmOutput=>bAlarmOutput , 
	bEnable:=bEnable AND mDevAlarmCheck(), 
	rProcessValue:=rProcessValue , 
	rSetPoint:=rSetpoint , 
	rDevLimit:=rDevLimitInternal , 
	bBlockHighAlarm:=bBlockHighAlarm , 
	bBlockLowAlarm:=bBlockLowAlarm );

	IF iStartSequence > 0 AND iStartSequence < 3 THEN
	 iStartSequenceInternal	 := 3 - iStartSequence;
	END_IF;

	fbSeqLink01(
	bEn:= bEnable, 
	udiSttCtrl:=iStartSequenceInternal , 
	udiIniSwiOvrDly_sec:= 5, 
	rX:= rProcessValue, 
	stSeqLink:=stSeqLink01 , 
	udiCurCtrl=> , 
	bSeqActv=> , 
	bNotRead=> , 
	bNoneOp=> , 
	udiRemTiIniSwiOvrDly_sec=> , 
	bErr=> , 
	sErrDescr=> );
	
	IF bBlockSequence1 THEN
		rTempMin := 0;
		rTempMax := 0;
	ELSE
		rTempMin := rMinSeq1;
		rTempMax := rMaxSeq1;
	END_IF
	rSetPointSequence1 := mCoolSetpointCheck(bActnSequence1);
	fbPidSeq[1](
	bEn:=bEnable , 
	rW:= rSetPointSequence1, 
	rX:=rProcessValue , 
	udiOpMode:= , 
	bActn:=bActnSequence1 , 
	rKp:= rKpSequence1, 
	udiTn_ms:=rKiSequence1*1000 , 
	udiTv_ms:=rDiSequence1*1000 , 
	udiTd_ms:=rFDiSequence1*1000 , 
	rYMax:=rTempMax , 
	rYMin:=rTempMin , 
	rNZ:= rDzSequence1, 
	udiCycCl:= , 
	bSync:= , 
	rSync:= , 
	rYSeqInit:= , 
	udiMyNum:= 2, 
	stSeqLink:=stSeqLink01 , 
	rY=> rOutputSequence1, 
	rE=> , 
	bErr=> , 
	sErrDescr=> );
	
	IF bBlockSequence2 THEN
		rTempMin := 0;
		rTempMax := 0;
	ELSE
		rTempMin := rMinSeq2;
		rTempMax := rMaxSeq2;
	END_IF
	rSetPointSequence2 := mCoolSetpointCheck(bActnSequence2);
	fbPidSeq[2](
	bEn:=bEnable , 
	rW:= rSetPointSequence2, 
	rX:= rProcessValue, 
	udiOpMode:= , 
	bActn:= bActnSequence2, 
	rKp:= rKpSequence2, 
	udiTn_ms:=rKiSequence2*1000 , 
	udiTv_ms:=rDiSequence2*1000  , 
	udiTd_ms:=rFDiSequence2*1000 , 
	rYMax:=rTempMax , 
	rYMin:=rTempMin , 
	rNZ:= rDzSequence2, 
	udiCycCl:= , 
	bSync:= , 
	rSync:= , 
	rYSeqInit:= , 
	udiMyNum:= 1, 
	stSeqLink:= stSeqLink01, 
	rY=> rOutputSequence2, 
	rE=> , 
	bErr=> , 
	sErrDescr=> );

// Publik metod för att kolla ifall det finns någon kylsekvens i regleringen. Kan exempelvis användas för att blockera högavvikelselarm vid hög utetemperatur då kylsekvens saknas.
METHOD PUBLIC mContainsCoolingSequence : BOOL
mContainsCoolingSequence := bActnSequence1 OR bActnSequence2;
END_METHOD

// Metod för att kolla ifall det är en kylsekvens och om det i sådant fall är något knutet på rCoolSetpoint
METHOD PRIVATE mCoolSetpointCheck : REAL // Valt börvärde
VAR_INPUT
	bActn : BOOL; // Koll av gångriktning
END_VAR
IF NOT bActn THEN
	mCoolSetpointCheck := rSetpoint;
ELSE
	IF __ISVALIDREF(rCoolSetpoint) THEN 
		mCoolSetpointCheck := rCoolSetpoint;
	ELSE
		mCoolSetpointCheck := rSetpoint;
	END_IF
END_IF
END_METHOD

// Kolla ifall något är knutet på inputen rDevLimit. Är inget knutet där inaktiveras avvikelselarmet.
METHOD PRIVATE mDevAlarmCheck : BOOL // Valt börvärde
IF __ISVALIDREF(rDevLimit) THEN 
	mDevAlarmCheck := TRUE;
	rDevLimitInternal := rDevLimit;
ELSE
	mDevAlarmCheck := FALSE;
END_IF
END_METHOD

END_FUNCTION_BLOCK

// oaksLibrary/Regulatorer/fbSequenceController3Stages
// Pi-regulator 3-sekvens
{attribute 'initialize_on_call'}
FUNCTION_BLOCK fbSequenceController3Stages
VAR_INPUT
	bEnable : BOOL; // Aktiverar reglering
	rProcessValue : REAL; // Aktuellt Ärvärde 
	rSetpoint : REAL; // Aktuellt börvärde. Önskas separat kylbörvärde för kylsekvenser se inputen rCoolSetpoint.
	{attribute 'initialize_on_call'}
	rCoolSetpoint : REFERENCE TO REAL; //Om man önskar ha ett högre börvärde för kylsekvenser lägg denna här så väljs detta på de sekvenser där bActnSequenceX = TRUE. Lämnar man inputen tom körs rSetpoint på både kyl och värmesekvenser.
	rMinSeq1 : REAL := 0; 
	rMaxSeq1 : REAL := 100;
	bActnSequence1 : BOOL; // Gångriktning reglersekvens  (kylsekvens = TRUE)
	bBlockSequence1 : BOOL; // blockera denna sekvens kan användas exempelvis vid nattkyla
	rMinSeq2 : REAL := 0; 
	rMaxSeq2 : REAL := 100;
	bActnSequence2 : BOOL; // Gångriktning reglersekvens  (kylsekvens = TRUE)
	bBlockSequence2 : BOOL; // blockera denna sekvens kan användas exempelvis vid nattkyla
	rMinSeq3 : REAL := 0; 
	rMaxSeq3 : REAL := 100;
	bActnSequence3 : BOOL; // Gångriktning reglersekvens  (kylsekvens = TRUE)
	bBlockSequence3 : BOOL; // blockera denna sekvens kan användas exempelvis vid nattkyla
	rKpSequence1 : REAL; // Kp
	rKiSequence1 : UDINT; // Ki
	rDiSequence1 : UDINT; // D-tid (Derivata)
	rFDiSequence1 : UDINT; // Filter tid D (Derivata)
	rDzSequence1 : REAL :=0.1; //Dödzon
	rKpSequence2 : REAL; // Kp
	rKiSequence2 : UDINT; // Ki
	rDiSequence2 : UDINT; // D-tid (Derivata)
	rFDiSequence2 : UDINT; // Filter tid D (Derivata)
	rDzSequence2 : REAL :=0.1; //Dödzon
	rKpSequence3 : REAL; // Kp
	rKiSequence3 : UDINT; // Ki
	rDiSequence3 : UDINT; // D-tid (Derivata)
	rFDiSequence3 : UDINT; // Filter tid D (Derivata)
	rDzSequence3 : REAL :=0.1; //Dödzon
	iStartSequence : UDINT :=3; //Sekvens där regulator startar
	{attribute 'pingroup' := 'DeviationAlarm'}
	{attribute 'initialize_on_call'}
	rDevLimit : REFERENCE TO REAL := 0;
	{attribute 'pingroup' := 'DeviationAlarm'}
	bBlockHighAlarm : BOOL; // Blockera högtemplarm
	{attribute 'pingroup' := 'DeviationAlarm'}
	bBlockLowAlarm : BOOL; // Blockera lågtemplarm
	{attribute 'pingroup' := 'DeviationAlarm'}
	tAlarmDelay : TIME := T#5S; // larmfördröjning
END_VAR
VAR_OUTPUT
	rOutputSequence1 : REAL;  // regulatorsignal
	rOutputSequence2 : REAL;  // regulatorsignal
	rOutputSequence3 : REAL;  // regulatorsignal
	{attribute 'pingroup' := 'DeviationAlarm'}
	bAlarmOutput : BOOL; //larmutgång
END_VAR
VAR
	rDevLimitInternal : REAL;
	fbDevAlarmPV: fbDevAlarm;
	rSetPointSequence1,rSetPointSequence2,rSetPointSequence3 : REAL; 		

	rTempMin,rTempMax : REAL; // tempvariabel för blockering av sekvenser 
	fbSeqLink01: Tc3_BA_Common.FB_BA_SeqLink;
	stSeqLink01 : Tc3_BA_Common.ST_BA_SeqLink;
	fbPidSeq: ARRAY[1..3] OF Tc3_BA_Common.FB_BA_SeqCtrl;
	iStartSequenceInternal : UDINT := 3;
END_VAR

	fbDevAlarmPV(
	tAlarmDelay:=tAlarmDelay , 
	bAutoReset:=TRUE , 
	bAlarmOutput=>bAlarmOutput , 
	bEnable:=bEnable AND mDevAlarmCheck(), 
	rProcessValue:=rProcessValue , 
	rSetPoint:=rSetpoint , 
	rDevLimit:=rDevLimitInternal , 
	bBlockHighAlarm:=bBlockHighAlarm , 
	bBlockLowAlarm:=bBlockLowAlarm );

	IF iStartSequence > 0 AND iStartSequence < 4 THEN
	 iStartSequenceInternal	 := 4 - iStartSequence;
	END_IF;
		
	
	fbSeqLink01(
	bEn:= bEnable, 
	udiSttCtrl:= iStartSequenceInternal, 
	udiIniSwiOvrDly_sec:= 5, 
	rX:= rProcessValue, 
	stSeqLink:=stSeqLink01 , 
	udiCurCtrl=> , 
	bSeqActv=> , 
	bNotRead=> , 
	bNoneOp=> , 
	udiRemTiIniSwiOvrDly_sec=> , 
	bErr=> , 
	sErrDescr=> );
	
	IF bBlockSequence1 THEN
		rTempMin := 0;
		rTempMax := 0;
	ELSE
		rTempMin := rMinSeq1;
		rTempMax := rMaxSeq1;
	END_IF
	rSetPointSequence1 := mCoolSetpointCheck(bActnSequence1);
	fbPidSeq[1](
	bEn:=bEnable , 
	rW:= rSetPointSequence1, 
	rX:=rProcessValue , 
	udiOpMode:= , 
	bActn:=bActnSequence1 , 
	rKp:= rKpSequence1, 
	udiTn_ms:=rKiSequence1*1000 , 
	udiTv_ms:=rDiSequence1*1000 , 
	udiTd_ms:=rFDiSequence1*1000 , 
	rYMax:=rTempMax , 
	rYMin:= rTempMin, 
	rNZ:= rDzSequence1, 
	udiCycCl:= , 
	bSync:= , 
	rSync:= , 
	rYSeqInit:= , 
	udiMyNum:= 3, 
	stSeqLink:=stSeqLink01 , 
	rY=> rOutputSequence1, 
	rE=> , 
	bErr=> , 
	sErrDescr=> );
	
	IF bBlockSequence2 THEN
		rTempMin := 0;
		rTempMax := 0;
	ELSE
		rTempMin := rMinSeq2;
		rTempMax := rMaxSeq2;
	END_IF
	rSetPointSequence2 := mCoolSetpointCheck(bActnSequence2);
	fbPidSeq[2](
	bEn:=bEnable , 
	rW:= rSetPointSequence2, 
	rX:= rProcessValue, 
	udiOpMode:= , 
	bActn:= bActnSequence2, 
	rKp:= rKpSequence2, 
	udiTn_ms:=rKiSequence2*1000 , 
	udiTv_ms:=rDiSequence2*1000 , 
	udiTd_ms:=rFDiSequence2*1000 , 
	rYMax:= rTempMax, 
	rYMin:=rTempMin , 
	rNZ:= rDzSequence2, 
	udiCycCl:= , 
	bSync:= , 
	rSync:= , 
	rYSeqInit:= , 
	udiMyNum:= 2, 
	stSeqLink:= stSeqLink01, 
	rY=> rOutputSequence2, 
	rE=> , 
	bErr=> , 
	sErrDescr=> );
	
	IF bBlockSequence3 THEN
		rTempMin := 0;
		rTempMax := 0;
	ELSE
		rTempMin := rMinSeq3;
		rTempMax := rMaxSeq3;
	END_IF
	rSetPointSequence3 := mCoolSetpointCheck(bActnSequence3);
	fbPidSeq[3](
	bEn:=bEnable , 
	rW:= rSetPointSequence3, 
	rX:= rProcessValue, 
	udiOpMode:= , 
	bActn:= bActnSequence3, 
	rKp:= rKpSequence3, 
	udiTn_ms:=rKiSequence3*1000 , 
	udiTv_ms:=rDiSequence3*1000 , 
	udiTd_ms:=rFDiSequence3*1000 , 
	rYMax:=rTempMax , 
	rYMin:= rTempMin, 
	rNZ:= rDzSequence3, 
	udiCycCl:= , 
	bSync:= , 
	rSync:= , 
	rYSeqInit:= , 
	udiMyNum:= 1, 
	stSeqLink:= stSeqLink01, 
	rY=> rOutputSequence3, 
	rE=> , 
	bErr=> , 
	sErrDescr=> );

// Publik metod för att kolla ifall det finns någon kylsekvens i regleringen. Kan exempelvis användas för att blockera högavvikelselarm vid hög utetemperatur då kylsekvens saknas.
METHOD PUBLIC mContainsCoolingSequence : BOOL
mContainsCoolingSequence := bActnSequence1 OR bActnSequence2 OR bActnSequence3;
END_METHOD

// Metod för att kolla ifall det är en kylsekvens och om det i sådant fall är något knutet på rCoolSetpoint
METHOD PRIVATE mCoolSetpointCheck : REAL // Valt börvärde
VAR_INPUT
	bActn : BOOL; // Koll av gångriktning
END_VAR
IF NOT bActn THEN
	mCoolSetpointCheck := rSetpoint;
ELSE
	IF __ISVALIDREF(rCoolSetpoint) THEN 
		mCoolSetpointCheck := rCoolSetpoint;
	ELSE
		mCoolSetpointCheck := rSetpoint;
	END_IF
END_IF
END_METHOD

// Kolla ifall något är knutet på inputen rDevLimit. Är inget knutet där inaktiveras avvikelselarmet.
METHOD PRIVATE mDevAlarmCheck : BOOL // Valt börvärde
IF __ISVALIDREF(rDevLimit) THEN 
	mDevAlarmCheck := TRUE;
	rDevLimitInternal := rDevLimit;
ELSE
	mDevAlarmCheck := FALSE;
END_IF
END_METHOD

END_FUNCTION_BLOCK

// oaksLibrary/Regulatorer/fbSequenceController4Stages
// Pi-regulator 4-sekvens
{attribute 'initialize_on_call'}
FUNCTION_BLOCK fbSequenceController4Stages
VAR_INPUT
	bEnable : BOOL; // Aktiverar reglering
	rProcessValue : REAL; // Aktuellt Ärvärde 
	rSetpoint : REAL; // Aktuellt börvärde. Önskas separat kylbörvärde för kylsekvenser se inputen rCoolSetpoint.
	{attribute 'initialize_on_call'}
	rCoolSetpoint : REFERENCE TO REAL; //Om man önskar ha ett högre börvärde för kylsekvenser lägg denna här så väljs detta på de sekvenser där bActnSequenceX = TRUE. Lämnar man inputen tom körs rSetpoint på både kyl och värmesekvenser.
	rMinSeq1 : REAL := 0; 
	rMaxSeq1 : REAL := 100;
	bActnSequence1 : BOOL; // Gångriktning reglersekvens  (kylsekvens = TRUE)
	bBlockSequence1 : BOOL; // blockera denna sekvens kan användas exempelvis vid nattkyla
	rMinSeq2 : REAL := 0; 
	rMaxSeq2 : REAL := 100;
	bActnSequence2 : BOOL; // Gångriktning reglersekvens  (kylsekvens = TRUE)
	bBlockSequence2 : BOOL; // blockera denna sekvens kan användas exempelvis vid nattkyla
	rMinSeq3 : REAL := 0; 
	rMaxSeq3 : REAL := 100;
	bActnSequence3 : BOOL; // Gångriktning reglersekvens  (kylsekvens = TRUE)
	bBlockSequence3 : BOOL; // blockera denna sekvens kan användas exempelvis vid nattkyla
	rMinSeq4 : REAL := 0; 
	rMaxSeq4 : REAL := 100;
	bActnSequence4 : BOOL; // Gångriktning reglersekvens  (kylsekvens = TRUE)
	bBlockSequence4 : BOOL; // blockera denna sekvens kan användas exempelvis vid nattkyla
	rKpSequence1 : REAL; // Kp
	rKiSequence1 : UDINT; // Ki
	rDiSequence1 : UDINT; // D-tid (Derivata)
	rFDiSequence1 : UDINT; // Filter tid D (Derivata)
	rDzSequence1 : REAL :=0.1; //Dödzon
	rKpSequence2 : REAL; // Kp
	rKiSequence2 : UDINT; // Ki
	rDiSequence2 : UDINT; // D-tid (Derivata)
	rFDiSequence2 : UDINT; // Filter tid D (Derivata)
	rDzSequence2 : REAL :=0.1; //Dödzon
	rKpSequence3 : REAL; // Kp
	rKiSequence3 : UDINT; // Ki
	rDiSequence3 : UDINT; // D-tid (Derivata)
	rFDiSequence3 : UDINT; // Filter tid D (Derivata)
	rDzSequence3 : REAL :=0.1; //Dödzon
	rKpSequence4 : REAL; // Kp
	rKiSequence4 : UDINT; // Ki
	rDiSequence4 : UDINT; // D-tid (Derivata)
	rFDiSequence4 : UDINT; // Filter tid D (Derivata)
	rDzSequence4 : REAL :=0.1; //Dödzon
	iStartSequence : UDINT :=3; //Sekvens där regulator startar
	{attribute 'pingroup' := 'DeviationAlarm'}
	{attribute 'initialize_on_call'}
	rDevLimit : REFERENCE TO REAL := 0;
	{attribute 'pingroup' := 'DeviationAlarm'}
	bBlockHighAlarm : BOOL; // Blockera högtemplarm
	{attribute 'pingroup' := 'DeviationAlarm'}
	bBlockLowAlarm : BOOL; // Blockera lågtemplarm
	{attribute 'pingroup' := 'DeviationAlarm'}
	tAlarmDelay : TIME := T#5S; // larmfördröjning
END_VAR
VAR_OUTPUT
	rY : REAL; // Utsignal huvudregulator
	rOutputSequence1 : REAL;  // regulatorsignal
	rOutputSequence2 : REAL;  // regulatorsignal
	rOutputSequence3 : REAL;  // regulatorsignal
	rOutputSequence4 : REAL;  // regulatorsignal
	{attribute 'pingroup' := 'DeviationAlarm'}
	bAlarmOutput : BOOL; //larmutgång
END_VAR
VAR
	rDevLimitInternal : REAL;
	fbDevAlarmPV: fbDevAlarm;
	rSetPointSequence1,rSetPointSequence2,rSetPointSequence3,rSetPointSequence4 : REAL; 	
	rTempMin,rTempMax : REAL; // tempvariabel för blockering av sekvenser 
	fbSeqLink01: Tc3_BA_Common.FB_BA_SeqLink;
	stSeqLink01 : Tc3_BA_Common.ST_BA_SeqLink;
	fbPidSeq: ARRAY[1..4] OF Tc3_BA_Common.FB_BA_SeqCtrl;
	iStartSequenceInternal : UDINT := 3;
END_VAR

	fbDevAlarmPV(
	tAlarmDelay:=tAlarmDelay , 
	bAutoReset:=TRUE , 
	bAlarmOutput=>bAlarmOutput , 
	bEnable:=bEnable AND mDevAlarmCheck(), 
	rProcessValue:=rProcessValue , 
	rSetPoint:=rSetpoint , 
	rDevLimit:=rDevLimitInternal , 
	bBlockHighAlarm:=bBlockHighAlarm , 
	bBlockLowAlarm:=bBlockLowAlarm );

	IF iStartSequence > 0 AND iStartSequence < 5 THEN
	 iStartSequenceInternal	 := 5 - iStartSequence;
	END_IF;
		
	
	fbSeqLink01(
	bEn:= bEnable, 
	udiSttCtrl:= iStartSequenceInternal, 
	udiIniSwiOvrDly_sec:= 5, 
	rX:= rProcessValue, 
	stSeqLink:=stSeqLink01 , 
	udiCurCtrl=> , 
	bSeqActv=> , 
	bNotRead=> , 
	bNoneOp=> , 
	udiRemTiIniSwiOvrDly_sec=> , 
	bErr=> , 
	sErrDescr=> );
		
	IF bBlockSequence1 THEN
		rTempMin := 0;
		rTempMax := 0;
	ELSE
		rTempMin := rMinSeq1;
		rTempMax := rMaxSeq1;
	END_IF
	rSetPointSequence1 := mCoolSetpointCheck(bActnSequence1);
	fbPidSeq[1](
	bEn:=bEnable , 
	rW:= rSetPointSequence1, 
	rX:=rProcessValue , 
	udiOpMode:= , 
	bActn:=bActnSequence1 , 
	rKp:= rKpSequence1, 
	udiTn_ms:=rKiSequence1*1000 , 
	udiTv_ms:=rDiSequence1*1000 , 
	udiTd_ms:=rFDiSequence1*1000 , 
	rYMax:=rTempMax , 
	rYMin:=rTempMin, 
	rNZ:= rDzSequence1, 
	udiCycCl:= , 
	bSync:= , 
	rSync:= , 
	rYSeqInit:= , 
	udiMyNum:= 4, 
	stSeqLink:=stSeqLink01 , 
	rY=> rOutputSequence1, 
	rE=> , 
	bErr=> , 
	sErrDescr=> );
	
	IF bBlockSequence2 THEN
		rTempMin := 0;
		rTempMax := 0;
	ELSE
		rTempMin := rMinSeq2;
		rTempMax := rMaxSeq2;
	END_IF
	rSetPointSequence2 := mCoolSetpointCheck(bActnSequence2);
	fbPidSeq[2](
	bEn:=bEnable , 
	rW:= rSetPointSequence2, 
	rX:= rProcessValue, 
	udiOpMode:= , 
	bActn:= bActnSequence2, 
	rKp:= rKpSequence2, 
	udiTn_ms:=rKiSequence2*1000 , 
	udiTv_ms:=rDiSequence2*1000 , 
	udiTd_ms:=rFDiSequence2*1000 , 
	rYMax:= rTempMax, 
	rYMin:=rTempMin , 
	rNZ:= rDzSequence2, 
	udiCycCl:= , 
	bSync:= , 
	rSync:= , 
	rYSeqInit:= , 
	udiMyNum:= 3, 
	stSeqLink:= stSeqLink01, 
	rY=> rOutputSequence2, 
	rE=> , 
	bErr=> , 
	sErrDescr=> );
	
	IF bBlockSequence3 THEN
		rTempMin := 0;
		rTempMax := 0;
	ELSE
		rTempMin := rMinSeq3;
		rTempMax := rMaxSeq3;
	END_IF
	rSetPointSequence3 := mCoolSetpointCheck(bActnSequence3);
	fbPidSeq[3](
	bEn:=bEnable , 
	rW:= rSetPointSequence3, 
	rX:= rProcessValue, 
	udiOpMode:= , 
	bActn:= bActnSequence3, 
	rKp:= rKpSequence3, 
	udiTn_ms:=rKiSequence3*1000 , 
	udiTv_ms:=rDiSequence3*1000 , 
	udiTd_ms:=rFDiSequence3*1000 , 
	rYMax:=rTempMax , 
	rYMin:= rTempMin, 
	rNZ:= rDzSequence3, 
	udiCycCl:= , 
	bSync:= , 
	rSync:= , 
	rYSeqInit:= , 
	udiMyNum:= 2, 
	stSeqLink:= stSeqLink01, 
	rY=> rOutputSequence3, 
	rE=> , 
	bErr=> , 
	sErrDescr=> );
	
	IF bBlockSequence4 THEN
		rTempMin := 0;
		rTempMax := 0;
	ELSE
		rTempMin := rMinSeq4;
		rTempMax := rMaxSeq4;
	END_IF
	rSetPointSequence4 := mCoolSetpointCheck(bActnSequence4);
	fbPidSeq[4](
	bEn:=bEnable , 
	rW:= rSetPointSequence4, 
	rX:= rProcessValue, 
	udiOpMode:= , 
	bActn:= bActnSequence4, 
	rKp:= rKpSequence4, 
	udiTn_ms:=rKiSequence4*1000 , 
	udiTv_ms:=rDiSequence4*1000 , 
	udiTd_ms:=rFDiSequence4*1000 , 
	rYMax:=rTempMax , 
	rYMin:= rTempMin, 
	rNZ:= rDzSequence4, 
	udiCycCl:= , 
	bSync:= , 
	rSync:= , 
	rYSeqInit:= , 
	udiMyNum:= 1, 
	stSeqLink:= stSeqLink01, 
	rY=> rOutputSequence4, 
	rE=> , 
	bErr=> , 
	sErrDescr=> );

// Publik metod för att kolla ifall det finns någon kylsekvens i regleringen. Kan exempelvis användas för att blockera högavvikelselarm vid hög utetemperatur då kylsekvens saknas.
METHOD PUBLIC mContainsCoolingSequence : BOOL
mContainsCoolingSequence := bActnSequence1 OR bActnSequence2 OR bActnSequence3 OR bActnSequence4;
END_METHOD

// Metod för att kolla ifall det är en kylsekvens och om det i sådant fall är något knutet på rCoolSetpoint
METHOD PRIVATE mCoolSetpointCheck : REAL // Valt börvärde
VAR_INPUT
	bActn : BOOL; // Koll av gångriktning
END_VAR
IF NOT bActn THEN
	mCoolSetpointCheck := rSetpoint;
ELSE
	IF __ISVALIDREF(rCoolSetpoint) THEN 
		mCoolSetpointCheck := rCoolSetpoint;
	ELSE
		mCoolSetpointCheck := rSetpoint;
	END_IF
END_IF
END_METHOD

// Kolla ifall något är knutet på inputen rDevLimit. Är inget knutet där inaktiveras avvikelselarmet.
METHOD PRIVATE mDevAlarmCheck : BOOL // Valt börvärde
IF __ISVALIDREF(rDevLimit) THEN 
	mDevAlarmCheck := TRUE;
	rDevLimitInternal := rDevLimit;
ELSE
	mDevAlarmCheck := FALSE;
END_IF
END_METHOD

END_FUNCTION_BLOCK

// oaksLibrary/Regulatorer/fbSequenceController5Stages
// Pi-regulator 5-sekvens
{attribute 'initialize_on_call'}
FUNCTION_BLOCK fbSequenceController5Stages
VAR_INPUT
	bEnable : BOOL; // Aktiverar reglering
	rProcessValue : REAL; // Aktuellt Ärvärde 
	rSetpoint : REAL; // Aktuellt börvärde. Önskas separat kylbörvärde för kylsekvenser se inputen rCoolSetpoint.
	{attribute 'initialize_on_call'}
	rCoolSetpoint : REFERENCE TO REAL; //Om man önskar ha ett högre börvärde för kylsekvenser lägg denna här så väljs detta på de sekvenser där bActnSequenceX = TRUE. Lämnar man inputen tom körs rSetpoint på både kyl och värmesekvenser.
	rMinSeq1 : REAL := 0; 
	rMaxSeq1 : REAL := 100;
	bActnSequence1 : BOOL; // Gångriktning reglersekvens  (kylsekvens = TRUE)
	bBlockSequence1 : BOOL; // blockera denna sekvens kan användas exempelvis vid nattkyla
	rMinSeq2 : REAL := 0; 
	rMaxSeq2 : REAL := 100;
	bActnSequence2 : BOOL; // Gångriktning reglersekvens  (kylsekvens = TRUE)
	bBlockSequence2 : BOOL; // blockera denna sekvens kan användas exempelvis vid nattkyla
	rMinSeq3 : REAL := 0; 
	rMaxSeq3 : REAL := 100;
	bActnSequence3 : BOOL; // Gångriktning reglersekvens  (kylsekvens = TRUE)
	bBlockSequence3 : BOOL; // blockera denna sekvens kan användas exempelvis vid nattkyla
	rMinSeq4 : REAL := 0; 
	rMaxSeq4 : REAL := 100;
	bActnSequence4 : BOOL; // Gångriktning reglersekvens  (kylsekvens = TRUE)
	bBlockSequence4 : BOOL; // blockera denna sekvens kan användas exempelvis vid nattkyla
	rMinSeq5 : REAL := 0; 
	rMaxSeq5 : REAL := 100;
	bActnSequence5 : BOOL; // Gångriktning reglersekvens  (kylsekvens = TRUE)
	bBlockSequence5 : BOOL; // blockera denna sekvens kan användas exempelvis vid nattkyla
	rKpSequence1 : REAL; // Kp
	rKiSequence1 : UDINT; // Ki
	rDiSequence1 : UDINT; // D-tid (Derivata)
	rFDiSequence1 : UDINT; // Filter tid D (Derivata)
	rDzSequence1 : REAL :=0.1; //Dödzon
	rKpSequence2 : REAL; // Kp
	rKiSequence2 : UDINT; // Ki
	rDiSequence2 : UDINT; // D-tid (Derivata)
	rFDiSequence2 : UDINT; // Filter tid D (Derivata)
	rDzSequence2 : REAL :=0.1; //Dödzon
	rKpSequence3 : REAL; // Kp
	rKiSequence3 : UDINT; // Ki
	rDiSequence3 : UDINT; // D-tid (Derivata)
	rFDiSequence3 : UDINT; // Filter tid D (Derivata)
	rDzSequence3 : REAL :=0.1; //Dödzon
	rKpSequence4 : REAL; // Kp
	rKiSequence4 : UDINT; // Ki
	rDiSequence4 : UDINT; // D-tid (Derivata)
	rFDiSequence4 : UDINT; // Filter tid D (Derivata)
	rDzSequence4 : REAL :=0.1; //Dödzon
	rKpSequence5 : REAL; // Kp
	rKiSequence5 : UDINT; // Ki
	rDiSequence5 : UDINT; // D-tid (Derivata)
	rDzSequence5 : REAL :=0.1; //Dödzon
	rFDiSequence5 : UDINT; // Filter tid D (Derivata)
	iStartSequence : UDINT :=3; //Sekvens där regulator startar
	{attribute 'pingroup' := 'DeviationAlarm'}
	{attribute 'initialize_on_call'}
	rDevLimit : REFERENCE TO REAL := 0;
	{attribute 'pingroup' := 'DeviationAlarm'}
	bBlockHighAlarm : BOOL; // Blockera högtemplarm
	{attribute 'pingroup' := 'DeviationAlarm'}
	bBlockLowAlarm : BOOL; // Blockera lågtemplarm
	{attribute 'pingroup' := 'DeviationAlarm'}
	tAlarmDelay : TIME := T#5S; // larmfördröjning
END_VAR
VAR_OUTPUT
	rY : REAL; // Utsignal huvudregulator
	rOutputSequence1 : REAL;  // regulatorsignal
	rOutputSequence2 : REAL;  // regulatorsignal
	rOutputSequence3 : REAL;  // regulatorsignal
	rOutputSequence4 : REAL;  // regulatorsignal
	rOutputSequence5 : REAL;  // regulatorsignal
	{attribute 'pingroup' := 'DeviationAlarm'}
	bAlarmOutput : BOOL; //larmutgång
END_VAR
VAR
	rDevLimitInternal : REAL;
	fbDevAlarmPV: fbDevAlarm;
	rSetPointSequence1,rSetPointSequence2,rSetPointSequence3,rSetPointSequence4,rSetPointSequence5 : REAL; 	
	rTempMin,rTempMax : REAL; // tempvariabel för blockering av sekvenser 
	fbSeqLink01: Tc3_BA_Common.FB_BA_SeqLink;
	stSeqLink01 : Tc3_BA_Common.ST_BA_SeqLink;
	fbPidSeq: ARRAY[1..5] OF Tc3_BA_Common.FB_BA_SeqCtrl;
	iStartSequenceInternal : UDINT := 3;
END_VAR

	fbDevAlarmPV(
	tAlarmDelay:=tAlarmDelay , 
	bAutoReset:=TRUE , 
	bAlarmOutput=>bAlarmOutput , 
	bEnable:=bEnable AND mDevAlarmCheck() , 
	rProcessValue:=rProcessValue , 
	rSetPoint:=rSetpoint , 
	rDevLimit:=rDevLimitInternal , 
	bBlockHighAlarm:=bBlockHighAlarm , 
	bBlockLowAlarm:=bBlockLowAlarm );

	IF iStartSequence > 0 AND iStartSequence < 5 THEN
	 iStartSequenceInternal	 := 5 - iStartSequence;
	END_IF;
		
	
	fbSeqLink01(
	bEn:= bEnable, 
	udiSttCtrl:= iStartSequenceInternal, 
	udiIniSwiOvrDly_sec:= 5, 
	rX:= rProcessValue, 
	stSeqLink:=stSeqLink01 , 
	udiCurCtrl=> , 
	bSeqActv=> , 
	bNotRead=> , 
	bNoneOp=> , 
	udiRemTiIniSwiOvrDly_sec=> , 
	bErr=> , 
	sErrDescr=> );
		
	IF bBlockSequence1 THEN
		rTempMin := 0;
		rTempMax := 0;
	ELSE
		rTempMin := rMinSeq1;
		rTempMax := rMaxSeq1;
	END_IF
	rSetPointSequence1 := mCoolSetpointCheck(bActnSequence1);
	fbPidSeq[1](
	bEn:=bEnable , 
	rW:= rSetPointSequence1, 
	rX:=rProcessValue , 
	udiOpMode:= , 
	bActn:=bActnSequence1 , 
	rKp:= rKpSequence1, 
	udiTn_ms:=rKiSequence1*1000 , 
	udiTv_ms:=rDiSequence1*1000 , 
	udiTd_ms:=rFDiSequence1*1000 , 
	rYMax:=rTempMax , 
	rYMin:=rTempMin, 
	rNZ:= rDzSequence1, 
	udiCycCl:= , 
	bSync:= , 
	rSync:= , 
	rYSeqInit:= , 
	udiMyNum:= 5, 
	stSeqLink:=stSeqLink01 , 
	rY=> rOutputSequence1, 
	rE=> , 
	bErr=> , 
	sErrDescr=> );
	
	IF bBlockSequence2 THEN
		rTempMin := 0;
		rTempMax := 0;
	ELSE
		rTempMin := rMinSeq2;
		rTempMax := rMaxSeq2;
	END_IF
	rSetPointSequence2 := mCoolSetpointCheck(bActnSequence2);
	fbPidSeq[2](
	bEn:=bEnable , 
	rW:= rSetPointSequence2, 
	rX:= rProcessValue, 
	udiOpMode:= , 
	bActn:= bActnSequence2, 
	rKp:= rKpSequence2, 
	udiTn_ms:=rKiSequence2*1000 , 
	udiTv_ms:=rDiSequence2*1000 , 
	udiTd_ms:=rFDiSequence2*1000 , 
	rYMax:= rTempMax, 
	rYMin:=rTempMin , 
	rNZ:= rDzSequence2, 
	udiCycCl:= , 
	bSync:= , 
	rSync:= , 
	rYSeqInit:= , 
	udiMyNum:= 4, 
	stSeqLink:= stSeqLink01, 
	rY=> rOutputSequence2, 
	rE=> , 
	bErr=> , 
	sErrDescr=> );
	
	IF bBlockSequence3 THEN
		rTempMin := 0;
		rTempMax := 0;
	ELSE
		rTempMin := rMinSeq3;
		rTempMax := rMaxSeq3;
	END_IF
	rSetPointSequence3 := mCoolSetpointCheck(bActnSequence3);
	fbPidSeq[3](
	bEn:=bEnable , 
	rW:= rSetPointSequence3, 
	rX:= rProcessValue, 
	udiOpMode:= , 
	bActn:= bActnSequence3, 
	rKp:= rKpSequence3, 
	udiTn_ms:=rKiSequence3*1000 , 
	udiTv_ms:=rDiSequence3*1000 , 
	udiTd_ms:=rFDiSequence3*1000 , 
	rYMax:=rTempMax , 
	rYMin:= rTempMin, 
	rNZ:= rDzSequence3, 
	udiCycCl:= , 
	bSync:= , 
	rSync:= , 
	rYSeqInit:= , 
	udiMyNum:= 3, 
	stSeqLink:= stSeqLink01, 
	rY=> rOutputSequence3, 
	rE=> , 
	bErr=> , 
	sErrDescr=> );
	
	IF bBlockSequence4 THEN
		rTempMin := 0;
		rTempMax := 0;
	ELSE
		rTempMin := rMinSeq4;
		rTempMax := rMaxSeq4;
	END_IF
	rSetPointSequence4 := mCoolSetpointCheck(bActnSequence4);
	fbPidSeq[4](
	bEn:=bEnable , 
	rW:= rSetPointSequence4, 
	rX:= rProcessValue, 
	udiOpMode:= , 
	bActn:= bActnSequence4, 
	rKp:= rKpSequence4, 
	udiTn_ms:=rKiSequence4*1000 , 
	udiTv_ms:=rDiSequence4*1000 , 
	udiTd_ms:=rFDiSequence4*1000 , 
	rYMax:=rTempMax , 
	rYMin:= rTempMin, 
	rNZ:= rDzSequence4, 
	udiCycCl:= , 
	bSync:= , 
	rSync:= , 
	rYSeqInit:= , 
	udiMyNum:= 2, 
	stSeqLink:= stSeqLink01, 
	rY=> rOutputSequence4, 
	rE=> , 
	bErr=> , 
	sErrDescr=> );
	
	IF bBlockSequence5 THEN
		rTempMin := 0;
		rTempMax := 0;
	ELSE
		rTempMin := rMinSeq5;
		rTempMax := rMaxSeq5;
	END_IF
	rSetPointSequence5 := mCoolSetpointCheck(bActnSequence5);
	fbPidSeq[5](
	bEn:=bEnable , 
	rW:= rSetPointSequence5, 
	rX:= rProcessValue, 
	udiOpMode:= , 
	bActn:= bActnSequence5, 
	rKp:= rKpSequence5, 
	udiTn_ms:=rKiSequence5*1000 , 
	udiTv_ms:=rDiSequence5*1000 , 
	udiTd_ms:=rFDiSequence5*1000 , 
	rYMax:=rTempMax , 
	rYMin:= rTempMin, 
	rNZ:= rDzSequence5, 
	udiCycCl:= , 
	bSync:= , 
	rSync:= , 
	rYSeqInit:= , 
	udiMyNum:= 1, 
	stSeqLink:= stSeqLink01, 
	rY=> rOutputSequence5, 
	rE=> , 
	bErr=> , 
	sErrDescr=> );

// Publik metod för att kolla ifall det finns någon kylsekvens i regleringen. Kan exempelvis användas för att blockera högavvikelselarm vid hög utetemperatur då kylsekvens saknas.
METHOD PUBLIC mContainsCoolingSequence : BOOL
mContainsCoolingSequence := bActnSequence1 OR bActnSequence2 OR bActnSequence3 OR bActnSequence4 OR bActnSequence5;
END_METHOD

// Metod för att kolla ifall det är en kylsekvens och om det i sådant fall är något knutet på rCoolSetpoint
METHOD PRIVATE mCoolSetpointCheck : REAL // Valt börvärde
VAR_INPUT
	bActn : BOOL; // Koll av gångriktning
END_VAR
IF NOT bActn THEN
	mCoolSetpointCheck := rSetpoint;
ELSE
	IF __ISVALIDREF(rCoolSetpoint) THEN 
		mCoolSetpointCheck := rCoolSetpoint;
	ELSE
		mCoolSetpointCheck := rSetpoint;
	END_IF
END_IF
END_METHOD

// Kolla ifall något är knutet på inputen rDevLimit. Är inget knutet där inaktiveras avvikelselarmet.
METHOD PRIVATE mDevAlarmCheck : BOOL // Valt börvärde
IF __ISVALIDREF(rDevLimit) THEN 
	mDevAlarmCheck := TRUE;
	rDevLimitInternal := rDevLimit;
ELSE
	mDevAlarmCheck := FALSE;
END_IF
END_METHOD

END_FUNCTION_BLOCK

// oaksLibrary/Regulatorer/fbSequenceController6Stages
// Pi-regulator 5-sekvens
{attribute 'initialize_on_call'}
FUNCTION_BLOCK fbSequenceController6Stages
VAR_INPUT
	bEnable : BOOL; // Aktiverar reglering
	rProcessValue : REAL; // Aktuellt Ärvärde 
	rSetpoint : REAL; // Aktuellt börvärde. Önskas separat kylbörvärde för kylsekvenser se inputen rCoolSetpoint.
	{attribute 'initialize_on_call'}
	rCoolSetpoint : REFERENCE TO REAL; //Om man önskar ha ett högre börvärde för kylsekvenser lägg denna här så väljs detta på de sekvenser där bActnSequenceX = TRUE. Lämnar man inputen tom körs rSetpoint på både kyl och värmesekvenser.
	rMinSeq1 : REAL := 0; 
	rMaxSeq1 : REAL := 100;
	bActnSequence1 : BOOL; // Gångriktning reglersekvens  (kylsekvens = TRUE)
	bBlockSequence1 : BOOL; // blockera denna sekvens kan användas exempelvis vid nattkyla
	rMinSeq2 : REAL := 0; 
	rMaxSeq2 : REAL := 100;
	bActnSequence2 : BOOL; // Gångriktning reglersekvens  (kylsekvens = TRUE)
	bBlockSequence2 : BOOL; // blockera denna sekvens kan användas exempelvis vid nattkyla
	rMinSeq3 : REAL := 0; 
	rMaxSeq3 : REAL := 100;
	bActnSequence3 : BOOL; // Gångriktning reglersekvens  (kylsekvens = TRUE)
	bBlockSequence3 : BOOL; // blockera denna sekvens kan användas exempelvis vid nattkyla
	rMinSeq4 : REAL := 0; 
	rMaxSeq4 : REAL := 100;
	bActnSequence4 : BOOL; // Gångriktning reglersekvens  (kylsekvens = TRUE)
	bBlockSequence4 : BOOL; // blockera denna sekvens kan användas exempelvis vid nattkyla
	rMinSeq5 : REAL := 0; 
	rMaxSeq5 : REAL := 100;
	bActnSequence5 : BOOL; // Gångriktning reglersekvens  (kylsekvens = TRUE)
	bBlockSequence5 : BOOL; // blockera denna sekvens kan användas exempelvis vid nattkyla
	rMinSeq6 : REAL := 0; 
	rMaxSeq6 : REAL := 100;
	bActnSequence6 : BOOL; // Gångriktning reglersekvens  (kylsekvens = TRUE)
	bBlockSequence6 : BOOL; // blockera denna sekvens kan användas exempelvis vid nattkyla
	rKpSequence1 : REAL; // Kp
	rKiSequence1 : UDINT; // Ki
	rDiSequence1 : UDINT; // D-tid (Derivata)
	rFDiSequence1 : UDINT; // Filter tid D (Derivata)
	rDzSequence1 : REAL :=0.1; //Dödzon
	rKpSequence2 : REAL; // Kp
	rKiSequence2 : UDINT; // Ki
	rDiSequence2 : UDINT; // D-tid (Derivata)
	rFDiSequence2 : UDINT; // Filter tid D (Derivata)
	rDzSequence2 : REAL :=0.1; //Dödzon
	rKpSequence3 : REAL; // Kp
	rKiSequence3 : UDINT; // Ki
	rDiSequence3 : UDINT; // D-tid (Derivata)
	rFDiSequence3 : UDINT; // Filter tid D (Derivata)
	rDzSequence3 : REAL :=0.1; //Dödzon
	rKpSequence4 : REAL; // Kp
	rKiSequence4 : UDINT; // Ki
	rDiSequence4 : UDINT; // D-tid (Derivata)
	rFDiSequence4 : UDINT; // Filter tid D (Derivata)
	rDzSequence4 : REAL :=0.1; //Dödzon
	rKpSequence5 : REAL; // Kp
	rKiSequence5 : UDINT; // Ki
	rDiSequence5 : UDINT; // D-tid (Derivata)
	rFDiSequence5 : UDINT; // Filter tid D (Derivata)
	rDzSequence5 : REAL :=0.1; //Dödzon
	rKpSequence6 : REAL; // Kp
	rKiSequence6 : UDINT; // Ki
	rDiSequence6 : UDINT; // D-tid (Derivata)
	rFDiSequence6 : UDINT; // Filter tid D (Derivata)
	rDzSequence6 : REAL :=0.1; //Dödzon
	iStartSequence : UDINT :=3; //Sekvens där regulator startar
	{attribute 'pingroup' := 'DeviationAlarm'}
	{attribute 'initialize_on_call'}
	rDevLimit : REFERENCE TO REAL := 0;
	{attribute 'pingroup' := 'DeviationAlarm'}
	bBlockHighAlarm : BOOL; // Blockera högtemplarm
	{attribute 'pingroup' := 'DeviationAlarm'}
	bBlockLowAlarm : BOOL; // Blockera lågtemplarm
	{attribute 'pingroup' := 'DeviationAlarm'}
	tAlarmDelay : TIME := T#5S; // larmfördröjning
END_VAR
VAR_OUTPUT
	rY : REAL; // Utsignal huvudregulator
	rOutputSequence1 : REAL;  // regulatorsignal
	rOutputSequence2 : REAL;  // regulatorsignal
	rOutputSequence3 : REAL;  // regulatorsignal
	rOutputSequence4 : REAL;  // regulatorsignal
	rOutputSequence5 : REAL;  // regulatorsignal
	rOutputSequence6 : REAL;  // regulatorsignal
	{attribute 'pingroup' := 'DeviationAlarm'}
	bAlarmOutput : BOOL; //larmutgång
END_VAR
VAR
	rDevLimitInternal : REAL;
	fbDevAlarmPV: fbDevAlarm;
	rSetPointSequence1,rSetPointSequence2,rSetPointSequence3,rSetPointSequence4,rSetPointSequence5,rSetPointSequence6 : REAL; 	
	rTempMin,rTempMax : REAL; // tempvariabel för blockering av sekvenser 
	fbSeqLink01: Tc3_BA_Common.FB_BA_SeqLink;
	stSeqLink01 : Tc3_BA_Common.ST_BA_SeqLink;
	fbPidSeq: ARRAY[1..6] OF Tc3_BA_Common.FB_BA_SeqCtrl;
	iStartSequenceInternal : UDINT := 3;
END_VAR

	fbDevAlarmPV(
	tAlarmDelay:=tAlarmDelay , 
	bAutoReset:=TRUE , 
	bAlarmOutput=>bAlarmOutput , 
	bEnable:=bEnable AND mDevAlarmCheck() , 
	rProcessValue:=rProcessValue , 
	rSetPoint:=rSetpoint , 
	rDevLimit:=rDevLimitInternal , 
	bBlockHighAlarm:=bBlockHighAlarm , 
	bBlockLowAlarm:=bBlockLowAlarm );

	IF iStartSequence > 0 AND iStartSequence < 6 THEN
	 iStartSequenceInternal	 := 6 - iStartSequence;
	END_IF;
		
	
	fbSeqLink01(
	bEn:= bEnable, 
	udiSttCtrl:= iStartSequenceInternal, 
	udiIniSwiOvrDly_sec:= 5, 
	rX:= rProcessValue, 
	stSeqLink:=stSeqLink01 , 
	udiCurCtrl=> , 
	bSeqActv=> , 
	bNotRead=> , 
	bNoneOp=> , 
	udiRemTiIniSwiOvrDly_sec=> , 
	bErr=> , 
	sErrDescr=> );
		
	IF bBlockSequence1 THEN
		rTempMin := 0;
		rTempMax := 0;
	ELSE
		rTempMin := rMinSeq1;
		rTempMax := rMaxSeq1;
	END_IF
	rSetPointSequence1 := mCoolSetpointCheck(bActnSequence1);
	fbPidSeq[1](
	bEn:=bEnable , 
	rW:= rSetPointSequence1, 
	rX:=rProcessValue , 
	udiOpMode:= , 
	bActn:=bActnSequence1 , 
	rKp:= rKpSequence1, 
	udiTn_ms:=rKiSequence1*1000 , 
	udiTv_ms:=rDiSequence1*1000 , 
	udiTd_ms:=rFDiSequence1*1000 , 
	rYMax:=rTempMax , 
	rYMin:=rTempMin, 
	rNZ:= rDzSequence1, 
	udiCycCl:= , 
	bSync:= , 
	rSync:= , 
	rYSeqInit:= , 
	udiMyNum:= 6, 
	stSeqLink:=stSeqLink01 , 
	rY=> rOutputSequence1, 
	rE=> , 
	bErr=> , 
	sErrDescr=> );
	
	IF bBlockSequence2 THEN
		rTempMin := 0;
		rTempMax := 0;
	ELSE
		rTempMin := rMinSeq2;
		rTempMax := rMaxSeq2;
	END_IF
	rSetPointSequence2 := mCoolSetpointCheck(bActnSequence2);
	fbPidSeq[2](
	bEn:=bEnable , 
	rW:= rSetPointSequence2, 
	rX:= rProcessValue, 
	udiOpMode:= , 
	bActn:= bActnSequence2, 
	rKp:= rKpSequence2, 
	udiTn_ms:=rKiSequence2*1000 , 
	udiTv_ms:=rDiSequence2*1000 , 
	udiTd_ms:=rFDiSequence2*1000 , 
	rYMax:= rTempMax, 
	rYMin:=rTempMin , 
	rNZ:= rDzSequence2, 
	udiCycCl:= , 
	bSync:= , 
	rSync:= , 
	rYSeqInit:= , 
	udiMyNum:= 5, 
	stSeqLink:= stSeqLink01, 
	rY=> rOutputSequence2, 
	rE=> , 
	bErr=> , 
	sErrDescr=> );
	
	IF bBlockSequence3 THEN
		rTempMin := 0;
		rTempMax := 0;
	ELSE
		rTempMin := rMinSeq3;
		rTempMax := rMaxSeq3;
	END_IF
	rSetPointSequence3 := mCoolSetpointCheck(bActnSequence3);
	fbPidSeq[3](
	bEn:=bEnable , 
	rW:= rSetPointSequence3, 
	rX:= rProcessValue, 
	udiOpMode:= , 
	bActn:= bActnSequence3, 
	rKp:= rKpSequence3, 
	udiTn_ms:=rKiSequence3*1000 , 
	udiTv_ms:=rDiSequence3*1000 , 
	udiTd_ms:=rFDiSequence3*1000 , 
	rYMax:=rTempMax , 
	rYMin:= rTempMin, 
	rNZ:= rDzSequence3, 
	udiCycCl:= , 
	bSync:= , 
	rSync:= , 
	rYSeqInit:= , 
	udiMyNum:= 4, 
	stSeqLink:= stSeqLink01, 
	rY=> rOutputSequence3, 
	rE=> , 
	bErr=> , 
	sErrDescr=> );
	
	IF bBlockSequence4 THEN
		rTempMin := 0;
		rTempMax := 0;
	ELSE
		rTempMin := rMinSeq4;
		rTempMax := rMaxSeq4;
	END_IF
	rSetPointSequence4 := mCoolSetpointCheck(bActnSequence4);
	fbPidSeq[4](
	bEn:=bEnable , 
	rW:= rSetPointSequence4, 
	rX:= rProcessValue, 
	udiOpMode:= , 
	bActn:= bActnSequence4, 
	rKp:= rKpSequence4, 
	udiTn_ms:=rKiSequence4*1000 , 
	udiTv_ms:=rDiSequence4*1000 , 
	udiTd_ms:=rFDiSequence4*1000 , 
	rYMax:=rTempMax , 
	rYMin:= rTempMin, 
	rNZ:= rDzSequence4, 
	udiCycCl:= , 
	bSync:= , 
	rSync:= , 
	rYSeqInit:= , 
	udiMyNum:= 3, 
	stSeqLink:= stSeqLink01, 
	rY=> rOutputSequence4, 
	rE=> , 
	bErr=> , 
	sErrDescr=> );
	
	IF bBlockSequence5 THEN
		rTempMin := 0;
		rTempMax := 0;
	ELSE
		rTempMin := rMinSeq5;
		rTempMax := rMaxSeq5;
	END_IF
	rSetPointSequence5 := mCoolSetpointCheck(bActnSequence5);
	fbPidSeq[5](
	bEn:=bEnable , 
	rW:= rSetPointSequence5, 
	rX:= rProcessValue, 
	udiOpMode:= , 
	bActn:= bActnSequence5, 
	rKp:= rKpSequence5, 
	udiTn_ms:=rKiSequence5*1000 , 
	udiTv_ms:=rDiSequence5*1000 , 
	udiTd_ms:=rFDiSequence5*1000 , 
	rYMax:=rTempMax , 
	rYMin:= rTempMin, 
	rNZ:= rDzSequence5, 
	udiCycCl:= , 
	bSync:= , 
	rSync:= , 
	rYSeqInit:= , 
	udiMyNum:= 2, 
	stSeqLink:= stSeqLink01, 
	rY=> rOutputSequence5, 
	rE=> , 
	bErr=> , 
	sErrDescr=> );
	
	IF bBlockSequence6 THEN
		rTempMin := 0;
		rTempMax := 0;
	ELSE
		rTempMin := rMinSeq6;
		rTempMax := rMaxSeq6;
	END_IF
	rSetPointSequence6 := mCoolSetpointCheck(bActnSequence6);
	fbPidSeq[6](
	bEn:=bEnable , 
	rW:= rSetPointSequence6, 
	rX:= rProcessValue, 
	udiOpMode:= , 
	bActn:= bActnSequence6, 
	rKp:= rKpSequence6, 
	udiTn_ms:=rKiSequence6*1000 , 
	udiTv_ms:=rDiSequence6*1000 , 
	udiTd_ms:=rFDiSequence6*1000 , 
	rYMax:=rTempMax , 
	rYMin:= rTempMin, 
	rNZ:= rDzSequence6, 
	udiCycCl:= , 
	bSync:= , 
	rSync:= , 
	rYSeqInit:= , 
	udiMyNum:= 1, 
	stSeqLink:= stSeqLink01, 
	rY=> rOutputSequence6, 
	rE=> , 
	bErr=> , 
	sErrDescr=> );

// Publik metod för att kolla ifall det finns någon kylsekvens i regleringen. Kan exempelvis användas för att blockera högavvikelselarm vid hög utetemperatur då kylsekvens saknas.
METHOD PUBLIC mContainsCoolingSequence : BOOL
mContainsCoolingSequence := bActnSequence1 OR bActnSequence2 OR bActnSequence3 OR bActnSequence4 OR bActnSequence5;
END_METHOD

// Metod för att kolla ifall det är en kylsekvens och om det i sådant fall är något knutet på rCoolSetpoint
METHOD PRIVATE mCoolSetpointCheck : REAL // Valt börvärde
VAR_INPUT
	bActn : BOOL; // Koll av gångriktning
END_VAR
IF NOT bActn THEN
	mCoolSetpointCheck := rSetpoint;
ELSE
	IF __ISVALIDREF(rCoolSetpoint) THEN 
		mCoolSetpointCheck := rCoolSetpoint;
	ELSE
		mCoolSetpointCheck := rSetpoint;
	END_IF
END_IF
END_METHOD

// Kolla ifall något är knutet på inputen rDevLimit. Är inget knutet där inaktiveras avvikelselarmet.
METHOD PRIVATE mDevAlarmCheck : BOOL // Valt börvärde
IF __ISVALIDREF(rDevLimit) THEN 
	mDevAlarmCheck := TRUE;
	rDevLimitInternal := rDevLimit;
ELSE
	mDevAlarmCheck := FALSE;
END_IF
END_METHOD

END_FUNCTION_BLOCK

